	2: (* === Check loop *)
		IF NOT (MB_Lock OR MB_Start) THEN
			WHILE VarCnt<=(VARS_Max-1) AND VarSta=2 DO
				(* Check only active vars *)
				IF VARS[VarCnt].Variable<>0 THEN			(* "Variable" is a pointer to word, so if 0 no address *)
					(* Check var auto-refresh on timer checks *)
					IF VARS[VarCnt].Refresh_Time>0 AND VARS[VarCnt].Refresh_Cnt=0 THEN
						VARS[VarCnt].Refresh_Cnt:=VARS[VarCnt].Refresh_Time;
						VarSta:=3;
					END_IF
					(* Check refresh for change or request *)
					CASE VARS[VarCnt].FunCode OF
						5,6,15,16: (* Write functions *)
							IF VARS[VarCnt].Variable_Size=1 THEN
								IF VARS[VarCnt].Variable^<>VARS[VarCnt].Variable_Mirror THEN
									VARS[VarCnt].Variable_Mirror:=VARS[VarCnt].Variable^;
									VarSta:=3;
								END_IF
							ELSE
								IF VARS[VarCnt].Variable_Mirror<>0 THEN
									VARS[VarCnt].Variable_Mirror:=0;
									VarSta:=3;
								END_IF
							END_IF
						1,2,3,4: (* Read functions *)
							IF VARS[VarCnt].Variable_Mirror<>0 THEN
								VARS[VarCnt].Variable_Mirror:=0;
								VarSta:=3;
							END_IF
					END_CASE
				END_IF
				(* Process query *)
				IF VarSta=3 THEN
					MB_Lock:=TRUE;
					MB_Query.SlaveAddress:=VARS[VarCnt].SlaveAddress;
					MB_Query.FunctionCode:=VARS[VarCnt].FunCode;
					CASE VARS[VarCnt].FunCode OF
						16#5,16#6,16#F,16#10:
							MB_Query.Read_Quantity:=0;
							MB_Query.Read_StartAddress:=0;
							MB_Query.Write_StartAddress:=VARS[VarCnt].FunAddress;
							MB_Query.Write_Quantity:=VARS[VarCnt].Variable_Size;
							IF VARS[VarCnt].Variable_Size=200 THEN
								COPY_32SWAP16(VARS[VarCnt].Variable, ADR(MB_Query.Write_Data[0]));
							ELSIF VARS[VarCnt].Variable_Size>1 THEN
								MEMCPY(VARS[VarCnt].Variable, ADR(MB_Query.Write_Data[0]), 2*VARS[VarCnt].Variable_Size);
							ELSE
								MB_Query.Write_Data[0]:=VARS[VarCnt].Variable^;
							END_IF
						16#1,16#2,16#3,16#4:
							MB_Query.Read_StartAddress:=VARS[VarCnt].FunAddress;
							IF VARS[VarCnt].Variable_Size=200 THEN MB_Query.Read_Quantity:=2; ELSE		(* 200 -->> DWORD 32bits *)
							  MB_Query.Read_Quantity:=VARS[VarCnt].Variable_Size;
							END_IF
							MB_Query.Write_StartAddress:=0;
							MB_Query.Write_Quantity:=0;
					END_CASE
					VarRetry:=0;
					MB_Start:=TRUE;
				ELSE
					VarCnt:=VarCnt+1;
				END_IF
			END_WHILE
			(* Check loop completed -> no actions *)
			IF VarSta=2 THEN VarSta:=1; END_IF
		END_IF

	3: (* === Wait & process MB response *)
		IF NOT MB_Start THEN
			IF MB_MASTER.MB_Error=0 THEN
				CASE VARS[VarCnt].FunCode OF
					1,2,3,4:
						IF VARS[VarCnt].Variable_Size=200 THEN
							COPY_32SWAP16(ADR(MB_Resp.Data), VARS[VarCnt].Variable);
						ELSIF VARS[VarCnt].Variable_Size>1 THEN
							MEMCPY(ADR(MB_Resp.Data), VARS[VarCnt].Variable, 2*VARS[VarCnt].Variable_Size);
						ELSE
							VARS[VarCnt].Variable^:=MB_Resp.Data[0];
						END_IF
				END_CASE
				MB_Lock:=FALSE;
				(* Signal error recovery *)
				IF VARS_Alarm=TRUE AND VarCnt=VarAlarm THEN
					LogEv(EL_Wrn,EO_MODBUS,ID,5,'');
					VARS_Alarm:=FALSE;
				END_IF
				(* Next var *)
				VarCnt:=VarCnt+1;
				VarSta:=2;
			ELSE
				IF VarRetry<3 THEN
					VarRetry:=VarRetry+1;
					MB_Start:=TRUE;
				ELSE
					MB_Lock:=FALSE;
					(* Signal error *)
					IF VARS_Alarm=FALSE THEN
						LogEv(EL_Wrn,EO_MODBUS,ID,3,INT_TO_STRING(MB_MASTER.MB_Error));
						VARS_Alarm:=TRUE;
						VarAlarm:=VarCnt-1;
					END_IF
					(* Next var *)
					VarCnt:=VarCnt+1;
					VarSta:=2;
				END_IF
			END_IF
		END_IF

ELSE
	VarSta:=0;
END_CASE
END_ACTION

(* POU Plant_Objects/obj_HVAC_LENNOX_FGK190H2M_new, ST *)
FUNCTION_BLOCK obj_HVAC_LENNOX_FGK190H2M_new
VAR CONSTANT
	Default_SetPointCold	: WORD 	:= 220;
	Default_SetPointHeat	: WORD 	:= 190;
	Default_SetBmsTenv		: INT 	:= -999;
	Default_SetBmsRHenv		: WORD	:= 0;
	Default_SetBmsText		: INT	:= -999;
	Default_SetBmsRHext		: WORD	:= 0;
	Default_MinThrECO		: WORD 	:= 1000;
	Default_MaxThrECO		: WORD 	:= 1500;
END_VAR
VAR_INPUT
	(* Settings *)
	ID						: BYTE;
	ADDRESS					: BYTE:=31;

	(* Controls *)
	Refresh_Period			: TIME:=t#3m;
	Refresh_Auto			: BOOL:=TRUE; (* Enable automatic refresh *)
	Refresh_Now				: BOOL; 	  (* Force an immediate refresh *)

	(* HVAC inputs	*)
	SetPointColdDay			: WORD;	(* Refresh set point	*)
	SetPointHeatDay			: WORD;	(* Heat set point		*)

	SetBmsTenv				: INT	:= Default_SetBmsTenv;	(* Environment temperature set point	*)
	SetBmsRHenv				: WORD	:= Default_SetBmsRHenv;	(* Environment humidity set point	*)
	SetBmsText				: INT	:= Default_SetBmsText;	(* External temperature set point 	*)
	SetBmsRHext				: WORD	:= Default_SetBmsRHext;	(* External humidity set point 	*)

	OnOff					: BOOL;

	MinThrECO				: WORD;
	MaxThrECO				: WORD;

END_VAR
VAR_IN_OUT
	MODBUS			: obj_MODBUS;
END_VAR
VAR_OUTPUT
	(* Sono read-only tetto il mondo *)
	Data			: typ_MODBUS_HVAC_LENNOX_FGK190H2M_new;
	tmpData			: typ_MODBUS_HVAC_LENNOX_FGK190H2M_new;

	(* Status *)
	Status_Log		: BYTE;
	Status_Vis 		: DWORD;

END_VAR
VAR

	dly 		: TON := (PT:=t#5s);
	sta			: BYTE; 	(* Status *)
	retry		: BYTE;
	fModbusAlr	: BOOL;

	ModbusAlr	:	FLT_EVENT;
	Alr1		:	FLT_EVENT;
	Alr2		:	FLT_EVENT;
	Alr3		:	FLT_EVENT;
	Alr4		:	FLT_EVENT;
	Alr5		:	FLT_EVENT;
	Alr6		:	FLT_EVENT;
	Alr7		:	FLT_EVENT;

	OldAlarm1	:	WORD;
	OldAlarm2	:	WORD;
	OldAlarm3	:	WORD;
	OldAlarm4	:	WORD;
	OldAlarm5	:	WORD;
	OldAlarm6	:	WORD;
	OldAlarm7	:	WORD;

	ChangedBits	:	WORD;
	AlarmCtr	:	BYTE;

	s1			:	STRING;
END_VAR
(* Verify inputs are in the right range	*)
CheckInputs();

(* Call ModBus state machine	*)
Stm();

(* Check if an alarm occurs	*)
CheckAlarm();

IF AlarmCtr>0 THEN
	Status_Log 	:= 2;
	Status_Vis	:= COLOR_RED;
ELSE
	Status_Log	:= 0;
	Status_Vis	:= COLOR_GREEN;
END_IF
END_FUNCTION_BLOCK
ACTION AddLogData:
Logger.s1:=INSERT('&HVAC=',BYTE_TO_STRING(ID),4);
IF ID<10 THEN Logger.s1:=INSERT(Logger.s1,'0',4); END_IF

Logger.s1:=CONCAT(Logger.s1,INT_TO_STRING(Data.Tsend));					Logger.s1:=CONCAT(Logger.s1,';');
Logger.s1:=CONCAT(Logger.s1,INT_TO_STRING(Data.Treturn));				Logger.s1:=CONCAT(Logger.s1,';');
Logger.s1:=CONCAT(Logger.s1,WORD_TO_STRING(Data.AirDiffPressure));		Logger.s1:=CONCAT(Logger.s1,';');
Logger.s1:=CONCAT(Logger.s1,WORD_TO_STRING(Data.AirValve));				Logger.s1:=CONCAT(Logger.s1,';');
Logger.s1:=CONCAT(Logger.s1,WORD_TO_STRING(Data.AirGas));				Logger.s1:=CONCAT(Logger.s1,';');
Logger.s1:=CONCAT(Logger.s1,WORD_TO_STRING(Data.Triac));				Logger.s1:=CONCAT(Logger.s1,';');
Logger.s1:=CONCAT(Logger.s1,WORD_TO_STRING(Data.HWB));					Logger.s1:=CONCAT(Logger.s1,';');
Logger.s1:=CONCAT(Logger.s1,WORD_TO_STRING(Data.Humidifier));			Logger.s1:=CONCAT(Logger.s1,';');

(* Create boolean representation of status flag and convert it in string *)
(*s1:=BOOL_TO_STRING(Data.StatusFlag.0);
s1:=CONCAT(s1,BOOL_TO_STRING(Data.StatusFlag.1));
s1:=CONCAT(s1,BOOL_TO_STRING(Data.StatusFlag.2));
s1:=CONCAT(s1,BOOL_TO_STRING(Data.StatusFlag.3));
s1:=CONCAT(s1,BOOL_TO_STRING(Data.StatusFlag.4));
s1:=CONCAT(s1,BOOL_TO_STRING(Data.StatusFlag.5));
s1:=CONCAT(s1,BOOL_TO_STRING(Data.StatusFlag.6));
s1:=CONCAT(s1,BOOL_TO_STRING(Data.StatusFlag.7));
s1:=CONCAT(s1,BOOL_TO_STRING(Data.StatusFlag.8));
s1:=CONCAT(s1,BOOL_TO_STRING(Data.StatusFlag.9));
s1:=CONCAT(s1,BOOL_TO_STRING(Data.StatusFlag.10));
s1:=CONCAT(s1,BOOL_TO_STRING(Data.StatusFlag.11));
s1:=CONCAT(s1,BOOL_TO_STRING(Data.StatusFlag.12));
s1:=CONCAT(s1,BOOL_TO_STRING(Data.StatusFlag.13));*)
s1:=BOOL_TO_STRING(Data.StatusFlag.13);
s1:=CONCAT(s1,BOOL_TO_STRING(Data.StatusFlag.12));
s1:=CONCAT(s1,BOOL_TO_STRING(Data.StatusFlag.11));
s1:=CONCAT(s1,BOOL_TO_STRING(Data.StatusFlag.10));
s1:=CONCAT(s1,BOOL_TO_STRING(Data.StatusFlag.9));
s1:=CONCAT(s1,BOOL_TO_STRING(Data.StatusFlag.8));
s1:=CONCAT(s1,BOOL_TO_STRING(Data.StatusFlag.7));
s1:=CONCAT(s1,BOOL_TO_STRING(Data.StatusFlag.6));
s1:=CONCAT(s1,BOOL_TO_STRING(Data.StatusFlag.5));
s1:=CONCAT(s1,BOOL_TO_STRING(Data.StatusFlag.4));
s1:=CONCAT(s1,BOOL_TO_STRING(Data.StatusFlag.3));
s1:=CONCAT(s1,BOOL_TO_STRING(Data.StatusFlag.2));
s1:=CONCAT(s1,BOOL_TO_STRING(Data.StatusFlag.1));
s1:=CONCAT(s1,BOOL_TO_STRING(Data.StatusFlag.0));

Logger.s1:=CONCAT(Logger.s1,s1);										Logger.s1:=CONCAT(Logger.s1,';');

(* Add operation times *)
Logger.s1:=CONCAT(Logger.s1,DWORD_TO_STRING(Data.HourVent));			Logger.s1:=CONCAT(Logger.s1,';');
Logger.s1:=CONCAT(Logger.s1,DWORD_TO_STRING(Data.HourCir1Comp1));		Logger.s1:=CONCAT(Logger.s1,';');
Logger.s1:=CONCAT(Logger.s1,DWORD_TO_STRING(Data.HourCir1Comp2));		Logger.s1:=CONCAT(Logger.s1,';');
Logger.s1:=CONCAT(Logger.s1,DWORD_TO_STRING(Data.HourCir2Comp1));		Logger.s1:=CONCAT(Logger.s1,';');
Logger.s1:=CONCAT(Logger.s1,DWORD_TO_STRING(Data.HourCir2Comp2));		Logger.s1:=CONCAT(Logger.s1,';');

Logger.s1:=CONCAT(Logger.s1,BYTE_TO_STRING(Status_Log));
ADDSTRING(ADR(Logger.TData), ADR(Logger.s1), Logger.TLen);
END_ACTION
ACTION CheckAlarm:
(* Modbus alarm *)
ModbusAlr(IN:=fModbusAlr);

IF ModbusAlr.EVH THEN
	LogEv(EL_Wrn,EO_HVAC,ID,2,SEL(ModBus.MB_MASTER.MB_Error<>0,'0','1'));
	Status_Log := 1;
END_IF

IF ModbusAlr.EVL THEN Status_Log := 0; END_IF	(* If there is an alarm, "Status_Log" wil be overwritten and becomes 2 *)


(***	ALARM 1		***)
(* Verify if at least one bit has changed in register "Alarm 1"	*)
Alr1(IN:=(Data.Alarm1 <> OldAlarm1));

IF Alr1.EVH THEN
	(* Consider just bit(s) that has changed its value (indicated by a logical 1 in "ChangedBits")	*)
	ChangedBits:= Data.Alarm1 XOR OldAlarm1;

	IF ChangedBits.0 THEN
		IF Data.Alarm1.0 THEN LogEv(EL_Alarm,EO_HVAC,ID,3,'70');	AlarmCtr := AlarmCtr + 1;
		ELSE LogEv(EL_Log,EO_HVAC,ID,4,'70'); 						AlarmCtr := AlarmCtr - 1;	END_IF
	END_IF

	IF ChangedBits.1 THEN
		IF Data.Alarm1.1 THEN LogEv(EL_Alarm,EO_HVAC,ID,3,'71');	AlarmCtr := AlarmCtr + 1;
		ELSE LogEv(EL_Log,EO_HVAC,ID,4,'71'); 						AlarmCtr := AlarmCtr - 1;	END_IF
	END_IF

	IF ChangedBits.2 THEN
		IF Data.Alarm1.2 THEN LogEv(EL_Alarm,EO_HVAC,ID,3,'72');	AlarmCtr := AlarmCtr + 1;
		ELSE LogEv(EL_Log,EO_HVAC,ID,4,'72'); 						AlarmCtr := AlarmCtr - 1;	END_IF
	END_IF

	IF ChangedBits.3 THEN
		IF Data.Alarm1.3 THEN LogEv(EL_Alarm,EO_HVAC,ID,3,'9');		AlarmCtr := AlarmCtr + 1;
		ELSE LogEv(EL_Log,EO_HVAC,ID,4,'9'); 						AlarmCtr := AlarmCtr - 1;	END_IF
	END_IF

	IF ChangedBits.4 THEN
		IF Data.Alarm1.4 THEN LogEv(EL_Alarm,EO_HVAC,ID,3,'81');	AlarmCtr := AlarmCtr + 1;
		ELSE LogEv(EL_Log,EO_HVAC,ID,4,'81'); 						AlarmCtr := AlarmCtr - 1;	END_IF
	END_IF

	IF ChangedBits.5 THEN
		IF Data.Alarm1.5 THEN LogEv(EL_Alarm,EO_HVAC,ID,3,'82');	AlarmCtr := AlarmCtr + 1;
		ELSE LogEv(EL_Log,EO_HVAC,ID,4,'82'); 						AlarmCtr := AlarmCtr - 1;	END_IF
	END_IF

	IF ChangedBits.6 THEN
		IF Data.Alarm1.6 THEN LogEv(EL_Alarm,EO_HVAC,ID,3,'83');	AlarmCtr := AlarmCtr + 1;
		ELSE LogEv(EL_Log,EO_HVAC,ID,4,'83'); 						AlarmCtr := AlarmCtr - 1;	END_IF
	END_IF

	IF ChangedBits.7 THEN
		IF Data.Alarm1.7 THEN LogEv(EL_Alarm,EO_HVAC,ID,3,'85');	AlarmCtr := AlarmCtr + 1;
		ELSE LogEv(EL_Log,EO_HVAC,ID,4,'85'); 						AlarmCtr := AlarmCtr - 1;	END_IF
	END_IF

	IF ChangedBits.8 THEN
		IF Data.Alarm1.8 THEN LogEv(EL_Alarm,EO_HVAC,ID,3,'88');	AlarmCtr := AlarmCtr + 1;
		ELSE LogEv(EL_Log,EO_HVAC,ID,4,'88'); 						AlarmCtr := AlarmCtr - 1;	END_IF
	END_IF

	IF ChangedBits.9 THEN
		IF Data.Alarm1.9 THEN LogEv(EL_Alarm,EO_HVAC,ID,3,'22');	AlarmCtr := AlarmCtr + 1;
		ELSE LogEv(EL_Log,EO_HVAC,ID,4,'22'); 						AlarmCtr := AlarmCtr - 1;	END_IF
	END_IF

	IF ChangedBits.10 THEN
		IF Data.Alarm1.10 THEN LogEv(EL_Alarm,EO_HVAC,ID,3,'80');	AlarmCtr := AlarmCtr + 1;
		ELSE LogEv(EL_Log,EO_HVAC,ID,4,'80'); 						AlarmCtr := AlarmCtr - 1;	END_IF
	END_IF

	IF ChangedBits.11 THEN
		IF Data.Alarm1.11 THEN LogEv(EL_Alarm,EO_HVAC,ID,3,'73');	AlarmCtr := AlarmCtr + 1;
		ELSE LogEv(EL_Log,EO_HVAC,ID,4,'73');	 					AlarmCtr := AlarmCtr - 1;	END_IF
	END_IF

	IF ChangedBits.12 THEN
		IF Data.Alarm1.12 THEN LogEv(EL_Alarm,EO_HVAC,ID,3,'1');	AlarmCtr := AlarmCtr + 1;
		ELSE LogEv(EL_Log,EO_HVAC,ID,4,'1'); 						AlarmCtr := AlarmCtr - 1;	END_IF
	END_IF

	IF ChangedBits.13 THEN
		IF Data.Alarm1.13 THEN LogEv(EL_Alarm,EO_HVAC,ID,3,'91');	AlarmCtr := AlarmCtr + 1;
		ELSE LogEv(EL_Log,EO_HVAC,ID,4,'91'); 						AlarmCtr := AlarmCtr - 1;	END_IF
	END_IF

	IF ChangedBits.14 THEN
		IF Data.Alarm1.14 THEN LogEv(EL_Alarm,EO_HVAC,ID,3,'92');	AlarmCtr := AlarmCtr + 1;
		ELSE LogEv(EL_Log,EO_HVAC,ID,4,'92'); 						AlarmCtr := AlarmCtr - 1;	END_IF
	END_IF

	IF ChangedBits.15 THEN
		IF Data.Alarm1.15 THEN LogEv(EL_Alarm,EO_HVAC,ID,3,'99');	AlarmCtr := AlarmCtr + 1;
		ELSE LogEv(EL_Log,EO_HVAC,ID,4,'99'); 						AlarmCtr := AlarmCtr - 1;	END_IF
	END_IF

END_IF


(***	ALARM 2		***)
Alr2(IN:=(Data.Alarm2 <> OldAlarm2));

IF Alr2.EVH THEN

	ChangedBits:= Data.Alarm2 XOR OldAlarm2;

	IF ChangedBits.0 THEN
		IF Data.Alarm2.0 THEN LogEv(EL_Alarm,EO_HVAC,ID,3,'74');	AlarmCtr := AlarmCtr + 1;
		ELSE LogEv(EL_Log,EO_HVAC,ID,4,'74'); 						AlarmCtr := AlarmCtr - 1;	END_IF
	END_IF

	IF ChangedBits.1 THEN
		IF Data.Alarm2.1 THEN LogEv(EL_Alarm,EO_HVAC,ID,3,'93');	AlarmCtr := AlarmCtr + 1;
		ELSE LogEv(EL_Log,EO_HVAC,ID,4,'93'); 						AlarmCtr := AlarmCtr - 1;	END_IF
	END_IF

	IF ChangedBits.2 THEN
		IF Data.Alarm2.2 THEN LogEv(EL_Alarm,EO_HVAC,ID,3,'94');	AlarmCtr := AlarmCtr + 1;
		ELSE LogEv(EL_Log,EO_HVAC,ID,4,'94'); 						AlarmCtr := AlarmCtr - 1;	END_IF
	END_IF

	(* No bit3 for this register	*)

	IF ChangedBits.4 THEN
		IF Data.Alarm2.4 THEN LogEv(EL_Alarm,EO_HVAC,ID,3,'59');	AlarmCtr := AlarmCtr + 1;
		ELSE LogEv(EL_Log,EO_HVAC,ID,4,'59'); 						AlarmCtr := AlarmCtr - 1;	END_IF
	END_IF

	IF ChangedBits.5 THEN
		IF Data.Alarm2.5 THEN LogEv(EL_Alarm,EO_HVAC,ID,3,'56');	AlarmCtr := AlarmCtr + 1;
		ELSE LogEv(EL_Log,EO_HVAC,ID,4,'56'); 						AlarmCtr := AlarmCtr - 1;	END_IF
	END_IF

	IF ChangedBits.6 THEN
		IF Data.Alarm2.6 THEN LogEv(EL_Alarm,EO_HVAC,ID,3,'51');	AlarmCtr := AlarmCtr + 1;
		ELSE LogEv(EL_Log,EO_HVAC,ID,4,'51'); 						AlarmCtr := AlarmCtr - 1;	END_IF
	END_IF

	IF ChangedBits.7 THEN
		IF Data.Alarm2.7 THEN LogEv(EL_Alarm,EO_HVAC,ID,3,'52');	AlarmCtr := AlarmCtr + 1;
		ELSE LogEv(EL_Log,EO_HVAC,ID,4,'52'); 						AlarmCtr := AlarmCtr - 1;	END_IF
	END_IF

	(* No bit8 for this register	*)

	IF ChangedBits.9 THEN
		IF Data.Alarm2.9 THEN LogEv(EL_Alarm,EO_HVAC,ID,3,'13');	AlarmCtr := AlarmCtr + 1;
		ELSE LogEv(EL_Log,EO_HVAC,ID,4,'13'); 						AlarmCtr := AlarmCtr - 1;	END_IF
	END_IF

	IF ChangedBits.10 THEN
		IF Data.Alarm2.10 THEN LogEv(EL_Alarm,EO_HVAC,ID,3,'41');	AlarmCtr := AlarmCtr + 1;
		ELSE LogEv(EL_Log,EO_HVAC,ID,4,'41'); 						AlarmCtr := AlarmCtr - 1;	END_IF
	END_IF

	IF ChangedBits.11 THEN
		IF Data.Alarm2.11 THEN LogEv(EL_Alarm,EO_HVAC,ID,3,'11');	AlarmCtr := AlarmCtr + 1;
		ELSE LogEv(EL_Log,EO_HVAC,ID,4,'11'); 						AlarmCtr := AlarmCtr - 1;	END_IF
	END_IF

	IF ChangedBits.12 THEN
		IF Data.Alarm2.12 THEN LogEv(EL_Alarm,EO_HVAC,ID,3,'12');	AlarmCtr := AlarmCtr + 1;
		ELSE LogEv(EL_Log,EO_HVAC,ID,4,'12'); 						AlarmCtr := AlarmCtr - 1;	END_IF
	END_IF

	IF ChangedBits.13 THEN
		IF Data.Alarm2.13 THEN LogEv(EL_Alarm,EO_HVAC,ID,3,'14');	AlarmCtr := AlarmCtr + 1;
		ELSE LogEv(EL_Log,EO_HVAC,ID,4,'14'); 						AlarmCtr := AlarmCtr - 1;	END_IF
	END_IF

	IF ChangedBits.14 THEN
		IF Data.Alarm2.14 THEN LogEv(EL_Alarm,EO_HVAC,ID,3,'15');	AlarmCtr := AlarmCtr + 1;
		ELSE LogEv(EL_Log,EO_HVAC,ID,4,'15'); 						AlarmCtr := AlarmCtr - 1;	END_IF
	END_IF

	IF ChangedBits.15 THEN
		IF Data.Alarm2.15 THEN LogEv(EL_Alarm,EO_HVAC,ID,3,'16');	AlarmCtr := AlarmCtr + 1;
		ELSE LogEv(EL_Log,EO_HVAC,ID,4,'16'); 						AlarmCtr := AlarmCtr - 1;	END_IF
	END_IF

END_IF


(***	ALARM 3		***)
Alr3(IN:=(Data.Alarm3 <> OldAlarm3));

IF Alr3.EVH THEN

	ChangedBits:= Data.Alarm3 XOR OldAlarm3;

	IF ChangedBits.0 THEN
		IF Data.Alarm3.0 THEN LogEv(EL_Alarm,EO_HVAC,ID,3,'141');	AlarmCtr := AlarmCtr + 1;
		ELSE LogEv(EL_Log,EO_HVAC,ID,4,'141'); 						AlarmCtr := AlarmCtr - 1;	END_IF
	END_IF

	IF ChangedBits.1 THEN
		IF Data.Alarm3.1 THEN LogEv(EL_Alarm,EO_HVAC,ID,3,'142');	AlarmCtr := AlarmCtr + 1;
		ELSE LogEv(EL_Log,EO_HVAC,ID,4,'142'); 						AlarmCtr := AlarmCtr - 1;	END_IF
	END_IF

	IF ChangedBits.2 THEN
		IF Data.Alarm3.2 THEN LogEv(EL_Alarm,EO_HVAC,ID,3,'143');	AlarmCtr := AlarmCtr + 1;
		ELSE LogEv(EL_Log,EO_HVAC,ID,4,'143'); 						AlarmCtr := AlarmCtr - 1;	END_IF
	END_IF

	IF ChangedBits.3 THEN
		IF Data.Alarm3.3 THEN LogEv(EL_Alarm,EO_HVAC,ID,3,'144');	AlarmCtr := AlarmCtr + 1;
		ELSE LogEv(EL_Log,EO_HVAC,ID,4,'144'); 						AlarmCtr := AlarmCtr - 1;	END_IF
	END_IF

	IF ChangedBits.4 THEN
		IF Data.Alarm3.4 THEN LogEv(EL_Alarm,EO_HVAC,ID,3,'114');	AlarmCtr := AlarmCtr + 1;
		ELSE LogEv(EL_Log,EO_HVAC,ID,4,'114'); 						AlarmCtr := AlarmCtr - 1;	END_IF
	END_IF

	IF ChangedBits.5 THEN
		IF Data.Alarm3.5 THEN LogEv(EL_Alarm,EO_HVAC,ID,3,'115');	AlarmCtr := AlarmCtr + 1;
		ELSE LogEv(EL_Log,EO_HVAC,ID,4,'115'); 						AlarmCtr := AlarmCtr - 1;	END_IF
	END_IF

	IF ChangedBits.6 THEN
		IF Data.Alarm3.6 THEN LogEv(EL_Alarm,EO_HVAC,ID,3,'116');	AlarmCtr := AlarmCtr + 1;
		ELSE LogEv(EL_Log,EO_HVAC,ID,4,'116'); 						AlarmCtr := AlarmCtr - 1;	END_IF
	END_IF

	IF ChangedBits.7 THEN
		IF Data.Alarm3.7 THEN LogEv(EL_Alarm,EO_HVAC,ID,3,'117');	AlarmCtr := AlarmCtr + 1;
		ELSE LogEv(EL_Log,EO_HVAC,ID,4,'117'); 						AlarmCtr := AlarmCtr - 1;	END_IF
	END_IF

	IF ChangedBits.8 THEN
		IF Data.Alarm3.8 THEN LogEv(EL_Alarm,EO_HVAC,ID,3,'118');	AlarmCtr := AlarmCtr + 1;
		ELSE LogEv(EL_Log,EO_HVAC,ID,4,'118'); 						AlarmCtr := AlarmCtr - 1;	END_IF
	END_IF

	IF ChangedBits.9 THEN
		IF Data.Alarm3.9 THEN LogEv(EL_Alarm,EO_HVAC,ID,3,'132');	AlarmCtr := AlarmCtr + 1;
		ELSE LogEv(EL_Log,EO_HVAC,ID,4,'132'); 						AlarmCtr := AlarmCtr - 1;	END_IF
	END_IF

	IF ChangedBits.10 THEN
		IF Data.Alarm3.10 THEN LogEv(EL_Alarm,EO_HVAC,ID,3,'75');	AlarmCtr := AlarmCtr + 1;
		ELSE LogEv(EL_Log,EO_HVAC,ID,4,'75'); 						AlarmCtr := AlarmCtr - 1;	END_IF
	END_IF

	IF ChangedBits.11 THEN
		IF Data.Alarm3.11 THEN LogEv(EL_Alarm,EO_HVAC,ID,3,'102');	AlarmCtr := AlarmCtr + 1;
		ELSE LogEv(EL_Log,EO_HVAC,ID,4,'102'); 						AlarmCtr := AlarmCtr - 1;	END_IF
	END_IF

	IF ChangedBits.12 THEN
		IF Data.Alarm3.12 THEN LogEv(EL_Alarm,EO_HVAC,ID,3,'103');	AlarmCtr := AlarmCtr + 1;
		ELSE LogEv(EL_Log,EO_HVAC,ID,4,'103'); 						AlarmCtr := AlarmCtr - 1;	END_IF
	END_IF

	IF ChangedBits.13 THEN
		IF Data.Alarm3.13 THEN LogEv(EL_Alarm,EO_HVAC,ID,3,'86');	AlarmCtr := AlarmCtr + 1;
		ELSE LogEv(EL_Log,EO_HVAC,ID,4,'86'); 						AlarmCtr := AlarmCtr - 1;	END_IF
	END_IF

	IF ChangedBits.14 THEN
		IF Data.Alarm3.14 THEN LogEv(EL_Alarm,EO_HVAC,ID,3,'87');	AlarmCtr := AlarmCtr + 1;
		ELSE LogEv(EL_Log,EO_HVAC,ID,4,'87'); 						AlarmCtr := AlarmCtr - 1;	END_IF
	END_IF

	IF ChangedBits.15 THEN
		IF Data.Alarm3.15 THEN LogEv(EL_Alarm,EO_HVAC,ID,3,'101');	AlarmCtr := AlarmCtr + 1;
		ELSE LogEv(EL_Log,EO_HVAC,ID,4,'101'); 						AlarmCtr := AlarmCtr - 1;	END_IF
	END_IF

END_IF


(***	ALARM 4		***)
Alr4(IN:=(Data.Alarm4 <> OldAlarm4));

IF Alr4.EVH THEN

	ChangedBits:= Data.Alarm4 XOR OldAlarm4;

	IF ChangedBits.0 THEN
		IF Data.Alarm4.0 THEN LogEv(EL_Alarm,EO_HVAC,ID,3,'241');	AlarmCtr := AlarmCtr + 1;
		ELSE LogEv(EL_Log,EO_HVAC,ID,4,'241'); 						AlarmCtr := AlarmCtr - 1;	END_IF
	END_IF

	IF ChangedBits.1 THEN
		IF Data.Alarm4.1 THEN LogEv(EL_Alarm,EO_HVAC,ID,3,'242');	AlarmCtr := AlarmCtr + 1;
		ELSE LogEv(EL_Log,EO_HVAC,ID,4,'242'); 						AlarmCtr := AlarmCtr - 1;	END_IF
	END_IF

	IF ChangedBits.2 THEN
		IF Data.Alarm4.2 THEN LogEv(EL_Alarm,EO_HVAC,ID,3,'243');	AlarmCtr := AlarmCtr + 1;
		ELSE LogEv(EL_Log,EO_HVAC,ID,4,'243'); 						AlarmCtr := AlarmCtr - 1;	END_IF
	END_IF

	IF ChangedBits.3 THEN
		IF Data.Alarm4.3 THEN LogEv(EL_Alarm,EO_HVAC,ID,3,'244');	AlarmCtr := AlarmCtr + 1;
		ELSE LogEv(EL_Log,EO_HVAC,ID,4,'244'); 						AlarmCtr := AlarmCtr - 1;	END_IF
	END_IF

	IF ChangedBits.4 THEN
		IF Data.Alarm4.4 THEN LogEv(EL_Alarm,EO_HVAC,ID,3,'214');	AlarmCtr := AlarmCtr + 1;
		ELSE LogEv(EL_Log,EO_HVAC,ID,4,'214'); 						AlarmCtr := AlarmCtr - 1;	END_IF
	END_IF

	IF ChangedBits.5 THEN
		IF Data.Alarm4.5 THEN LogEv(EL_Alarm,EO_HVAC,ID,3,'215');	AlarmCtr := AlarmCtr + 1;
		ELSE LogEv(EL_Log,EO_HVAC,ID,4,'215'); 						AlarmCtr := AlarmCtr - 1;	END_IF
	END_IF

	IF ChangedBits.6 THEN
		IF Data.Alarm4.6 THEN LogEv(EL_Alarm,EO_HVAC,ID,3,'216');	AlarmCtr := AlarmCtr + 1;
		ELSE LogEv(EL_Log,EO_HVAC,ID,4,'216'); 						AlarmCtr := AlarmCtr - 1;	END_IF
	END_IF

	IF ChangedBits.7 THEN
		IF Data.Alarm4.7 THEN LogEv(EL_Alarm,EO_HVAC,ID,3,'217');	AlarmCtr := AlarmCtr + 1;
		ELSE LogEv(EL_Log,EO_HVAC,ID,4,'217'); 						AlarmCtr := AlarmCtr - 1;	END_IF
	END_IF

	IF ChangedBits.8 THEN
		IF Data.Alarm4.8 THEN LogEv(EL_Alarm,EO_HVAC,ID,3,'218');	AlarmCtr := AlarmCtr + 1;
		ELSE LogEv(EL_Log,EO_HVAC,ID,4,'218'); 						AlarmCtr := AlarmCtr - 1;	END_IF
	END_IF

	IF ChangedBits.9 THEN
		IF Data.Alarm4.9 THEN LogEv(EL_Alarm,EO_HVAC,ID,3,'232');	AlarmCtr := AlarmCtr + 1;
		ELSE LogEv(EL_Log,EO_HVAC,ID,4,'232'); 						AlarmCtr := AlarmCtr - 1;	END_IF
	END_IF

	IF ChangedBits.10 THEN
		IF Data.Alarm4.10 THEN LogEv(EL_Alarm,EO_HVAC,ID,3,'76');	AlarmCtr := AlarmCtr + 1;
		ELSE LogEv(EL_Log,EO_HVAC,ID,4,'76'); 						AlarmCtr := AlarmCtr - 1;	END_IF
	END_IF

	IF ChangedBits.11 THEN
		IF Data.Alarm4.11 THEN LogEv(EL_Alarm,EO_HVAC,ID,3,'202');	AlarmCtr := AlarmCtr + 1;
		ELSE LogEv(EL_Log,EO_HVAC,ID,4,'202'); 						AlarmCtr := AlarmCtr - 1;	END_IF
	END_IF

	IF ChangedBits.12 THEN
		IF Data.Alarm4.12 THEN LogEv(EL_Alarm,EO_HVAC,ID,3,'203');	AlarmCtr := AlarmCtr + 1;
		ELSE LogEv(EL_Log,EO_HVAC,ID,4,'203'); 						AlarmCtr := AlarmCtr - 1;	END_IF
	END_IF

	IF ChangedBits.13 THEN
		IF Data.Alarm4.13 THEN LogEv(EL_Alarm,EO_HVAC,ID,3,'2');	AlarmCtr := AlarmCtr + 1;
		ELSE LogEv(EL_Log,EO_HVAC,ID,4,'2'); 						AlarmCtr := AlarmCtr - 1;	END_IF
	END_IF

	IF ChangedBits.14 THEN
		IF Data.Alarm4.14 THEN LogEv(EL_Alarm,EO_HVAC,ID,3,'25');	AlarmCtr := AlarmCtr + 1;
		ELSE LogEv(EL_Log,EO_HVAC,ID,4,'25'); 						AlarmCtr := AlarmCtr - 1;	END_IF
	END_IF

	IF ChangedBits.15 THEN
		IF Data.Alarm4.15 THEN LogEv(EL_Alarm,EO_HVAC,ID,3,'26');	AlarmCtr := AlarmCtr + 1;
		ELSE LogEv(EL_Log,EO_HVAC,ID,4,'26'); 						AlarmCtr := AlarmCtr - 1;	END_IF
	END_IF

END_IF


(***	ALARM 5		***)
Alr5(IN:=(Data.Alarm5 <> OldAlarm5));

IF Alr5.EVH THEN

	ChangedBits:= Data.Alarm5 XOR OldAlarm5;

	IF ChangedBits.0 THEN
		IF Data.Alarm5.0 THEN LogEv(EL_Alarm,EO_HVAC,ID,3,'84');	AlarmCtr := AlarmCtr + 1;
		ELSE LogEv(EL_Log,EO_HVAC,ID,4,'84'); 						AlarmCtr := AlarmCtr - 1;	END_IF
	END_IF

	IF ChangedBits.1 THEN
		IF Data.Alarm5.1 THEN LogEv(EL_Alarm,EO_HVAC,ID,3,'23');	AlarmCtr := AlarmCtr + 1;
		ELSE LogEv(EL_Log,EO_HVAC,ID,4,'23'); 						AlarmCtr := AlarmCtr - 1;	END_IF
	END_IF

	IF ChangedBits.2 THEN
		IF Data.Alarm5.2 THEN LogEv(EL_Alarm,EO_HVAC,ID,3,'24');	AlarmCtr := AlarmCtr + 1;
		ELSE LogEv(EL_Log,EO_HVAC,ID,4,'24'); 						AlarmCtr := AlarmCtr - 1;	END_IF
	END_IF

	IF ChangedBits.3 THEN
		IF Data.Alarm5.3 THEN LogEv(EL_Alarm,EO_HVAC,ID,3,'32');	AlarmCtr := AlarmCtr + 1;
		ELSE LogEv(EL_Log,EO_HVAC,ID,4,'32'); 						AlarmCtr := AlarmCtr - 1;	END_IF
	END_IF

	IF ChangedBits.4 THEN
		IF Data.Alarm5.4 THEN LogEv(EL_Alarm,EO_HVAC,ID,3,'33');	AlarmCtr := AlarmCtr + 1;
		ELSE LogEv(EL_Log,EO_HVAC,ID,4,'33'); 						AlarmCtr := AlarmCtr - 1;	END_IF
	END_IF

	IF ChangedBits.5 THEN
		IF Data.Alarm5.5 THEN LogEv(EL_Alarm,EO_HVAC,ID,3,'21');	AlarmCtr := AlarmCtr + 1;
		ELSE LogEv(EL_Log,EO_HVAC,ID,4,'21'); 						AlarmCtr := AlarmCtr - 1;	END_IF
	END_IF

	IF ChangedBits.6 THEN
		IF Data.Alarm5.6 THEN LogEv(EL_Alarm,EO_HVAC,ID,3,'4');		AlarmCtr := AlarmCtr + 1;
		ELSE LogEv(EL_Log,EO_HVAC,ID,4,'4'); 						AlarmCtr := AlarmCtr - 1;	END_IF
	END_IF

	IF ChangedBits.7 THEN
		IF Data.Alarm5.7 THEN LogEv(EL_Alarm,EO_HVAC,ID,3,'5');		AlarmCtr := AlarmCtr + 1;
		ELSE LogEv(EL_Log,EO_HVAC,ID,4,'5'); 						AlarmCtr := AlarmCtr - 1;	END_IF
	END_IF

	IF ChangedBits.8 THEN
		IF Data.Alarm5.8 THEN LogEv(EL_Alarm,EO_HVAC,ID,3,'89');	AlarmCtr := AlarmCtr + 1;
		ELSE LogEv(EL_Log,EO_HVAC,ID,4,'89'); 						AlarmCtr := AlarmCtr - 1;	END_IF
	END_IF

	IF ChangedBits.9 THEN
		IF Data.Alarm5.9 THEN LogEv(EL_Alarm,EO_HVAC,ID,3,'29');	AlarmCtr := AlarmCtr + 1;
		ELSE LogEv(EL_Log,EO_HVAC,ID,4,'29'); 						AlarmCtr := AlarmCtr - 1;	END_IF
	END_IF

	IF ChangedBits.10 THEN
		IF Data.Alarm5.10 THEN LogEv(EL_Alarm,EO_HVAC,ID,3,'54');	AlarmCtr := AlarmCtr + 1;
		ELSE LogEv(EL_Log,EO_HVAC,ID,4,'54'); 						AlarmCtr := AlarmCtr - 1;	END_IF
	END_IF

	IF ChangedBits.11 THEN
		IF Data.Alarm5.11 THEN LogEv(EL_Alarm,EO_HVAC,ID,3,'31');	AlarmCtr := AlarmCtr + 1;
		ELSE LogEv(EL_Log,EO_HVAC,ID,4,'31'); 						AlarmCtr := AlarmCtr - 1;	END_IF
	END_IF

	(* No bit12 and bit13 for this register	*)

	IF ChangedBits.14 THEN
		IF Data.Alarm5.14 THEN LogEv(EL_Alarm,EO_HVAC,ID,3,'110');	AlarmCtr := AlarmCtr + 1;
		ELSE LogEv(EL_Log,EO_HVAC,ID,4,'110'); 						AlarmCtr := AlarmCtr - 1;	END_IF
	END_IF

	IF ChangedBits.15 THEN
		IF Data.Alarm5.15 THEN LogEv(EL_Alarm,EO_HVAC,ID,3,'210');	AlarmCtr := AlarmCtr + 1;
		ELSE LogEv(EL_Log,EO_HVAC,ID,4,'210'); 						AlarmCtr := AlarmCtr - 1;	END_IF
	END_IF

END_IF


(***	ALARM 6		***)
Alr6(IN:=(Data.Alarm6 <> OldAlarm6));

IF Alr6.EVH THEN

	ChangedBits:= Data.Alarm6 XOR OldAlarm6;

	IF ChangedBits.0 THEN
		IF Data.Alarm6.0 THEN LogEv(EL_Alarm,EO_HVAC,ID,3,'119');	AlarmCtr := AlarmCtr + 1;
		ELSE LogEv(EL_Log,EO_HVAC,ID,4,'119'); 						AlarmCtr := AlarmCtr - 1;	END_IF
	END_IF

	IF ChangedBits.1 THEN
		IF Data.Alarm6.1 THEN LogEv(EL_Alarm,EO_HVAC,ID,3,'129');	AlarmCtr := AlarmCtr + 1;
		ELSE LogEv(EL_Log,EO_HVAC,ID,4,'129');	 					AlarmCtr := AlarmCtr - 1;	END_IF
	END_IF

	IF ChangedBits.2 THEN
		IF Data.Alarm6.2 THEN LogEv(EL_Alarm,EO_HVAC,ID,3,'128');	AlarmCtr := AlarmCtr + 1;
		ELSE LogEv(EL_Log,EO_HVAC,ID,4,'128'); 						AlarmCtr := AlarmCtr - 1;	END_IF
	END_IF

	IF ChangedBits.3 THEN
		IF Data.Alarm6.3 THEN LogEv(EL_Alarm,EO_HVAC,ID,3,'127');	AlarmCtr := AlarmCtr + 1;
		ELSE LogEv(EL_Log,EO_HVAC,ID,4,'127'); 						AlarmCtr := AlarmCtr - 1;	END_IF
	END_IF

	IF ChangedBits.4 THEN
		IF Data.Alarm6.4 THEN LogEv(EL_Alarm,EO_HVAC,ID,3,'121');	AlarmCtr := AlarmCtr + 1;
		ELSE LogEv(EL_Log,EO_HVAC,ID,4,'121'); 						AlarmCtr := AlarmCtr - 1;	END_IF
	END_IF

	IF ChangedBits.5 THEN
		IF Data.Alarm6.5 THEN LogEv(EL_Alarm,EO_HVAC,ID,3,'122');	AlarmCtr := AlarmCtr + 1;
		ELSE LogEv(EL_Log,EO_HVAC,ID,4,'122'); 						AlarmCtr := AlarmCtr - 1;	END_IF
	END_IF

	IF ChangedBits.6 THEN
		IF Data.Alarm6.6 THEN LogEv(EL_Alarm,EO_HVAC,ID,3,'123');	AlarmCtr := AlarmCtr + 1;
		ELSE LogEv(EL_Log,EO_HVAC,ID,4,'123'); 						AlarmCtr := AlarmCtr - 1;	END_IF
	END_IF

	IF ChangedBits.7 THEN
		IF Data.Alarm6.7 THEN LogEv(EL_Alarm,EO_HVAC,ID,3,'124');	AlarmCtr := AlarmCtr + 1;
		ELSE LogEv(EL_Log,EO_HVAC,ID,4,'124'); 						AlarmCtr := AlarmCtr - 1;	END_IF
	END_IF

	IF ChangedBits.8 THEN
		IF Data.Alarm6.8 THEN LogEv(EL_Alarm,EO_HVAC,ID,3,'219');	AlarmCtr := AlarmCtr + 1;
		ELSE LogEv(EL_Log,EO_HVAC,ID,4,'219'); 						AlarmCtr := AlarmCtr - 1;	END_IF
	END_IF

	IF ChangedBits.9 THEN
		IF Data.Alarm6.9 THEN LogEv(EL_Alarm,EO_HVAC,ID,3,'229');	AlarmCtr := AlarmCtr + 1;
		ELSE LogEv(EL_Log,EO_HVAC,ID,4,'229'); 						AlarmCtr := AlarmCtr - 1;	END_IF
	END_IF

	IF ChangedBits.10 THEN
		IF Data.Alarm6.10 THEN LogEv(EL_Alarm,EO_HVAC,ID,3,'228');	AlarmCtr := AlarmCtr + 1;
		ELSE LogEv(EL_Log,EO_HVAC,ID,4,'228'); 						AlarmCtr := AlarmCtr - 1;	END_IF
	END_IF

	IF ChangedBits.11 THEN
		IF Data.Alarm6.11 THEN LogEv(EL_Alarm,EO_HVAC,ID,3,'227');	AlarmCtr := AlarmCtr + 1;
		ELSE LogEv(EL_Log,EO_HVAC,ID,4,'227'); 						AlarmCtr := AlarmCtr - 1;	END_IF
	END_IF

	IF ChangedBits.12 THEN
		IF Data.Alarm6.12 THEN LogEv(EL_Alarm,EO_HVAC,ID,3,'221');	AlarmCtr := AlarmCtr + 1;
		ELSE LogEv(EL_Log,EO_HVAC,ID,4,'221'); 						AlarmCtr := AlarmCtr - 1;	END_IF
	END_IF

	IF ChangedBits.13 THEN
		IF Data.Alarm6.13 THEN LogEv(EL_Alarm,EO_HVAC,ID,3,'222');	AlarmCtr := AlarmCtr + 1;
		ELSE LogEv(EL_Log,EO_HVAC,ID,4,'222');	 					AlarmCtr := AlarmCtr - 1;	END_IF
	END_IF

	IF ChangedBits.14 THEN
		IF Data.Alarm6.14 THEN LogEv(EL_Alarm,EO_HVAC,ID,3,'223');	AlarmCtr := AlarmCtr + 1;
		ELSE LogEv(EL_Log,EO_HVAC,ID,4,'223'); 						AlarmCtr := AlarmCtr - 1;	END_IF
	END_IF

	IF ChangedBits.15 THEN
		IF Data.Alarm6.15 THEN LogEv(EL_Alarm,EO_HVAC,ID,3,'224');	AlarmCtr := AlarmCtr + 1;
		ELSE LogEv(EL_Log,EO_HVAC,ID,4,'224'); 						AlarmCtr := AlarmCtr - 1;	END_IF
	END_IF

END_IF


(***	ALARM 7		***)
Alr7(IN:=(Data.Alarm7 <> OldAlarm7));

IF Alr7.EVH THEN

	ChangedBits:= Data.Alarm7 XOR OldAlarm7;

	IF ChangedBits.0 THEN
		IF Data.Alarm7.0 THEN LogEv(EL_Alarm,EO_HVAC,ID,3,'341');	AlarmCtr := AlarmCtr + 1;
		ELSE LogEv(EL_Log,EO_HVAC,ID,4,'341'); 						AlarmCtr := AlarmCtr - 1;	END_IF
	END_IF

	IF ChangedBits.1 THEN
		IF Data.Alarm7.1 THEN LogEv(EL_Alarm,EO_HVAC,ID,3,'342');	AlarmCtr := AlarmCtr + 1;
		ELSE LogEv(EL_Log,EO_HVAC,ID,4,'342'); 						AlarmCtr := AlarmCtr - 1;	END_IF
	END_IF

	IF ChangedBits.2 THEN
		IF Data.Alarm7.2 THEN LogEv(EL_Alarm,EO_HVAC,ID,3,'343');	AlarmCtr := AlarmCtr + 1;
		ELSE LogEv(EL_Log,EO_HVAC,ID,4,'343'); 						AlarmCtr := AlarmCtr - 1;	END_IF
	END_IF

	IF ChangedBits.3 THEN
		IF Data.Alarm7.3 THEN LogEv(EL_Alarm,EO_HVAC,ID,3,'344');	AlarmCtr := AlarmCtr + 1;
		ELSE LogEv(EL_Log,EO_HVAC,ID,4,'344'); 						AlarmCtr := AlarmCtr - 1;	END_IF
	END_IF

	IF ChangedBits.4 THEN
		IF Data.Alarm7.4 THEN LogEv(EL_Alarm,EO_HVAC,ID,3,'314');	AlarmCtr := AlarmCtr + 1;
		ELSE LogEv(EL_Log,EO_HVAC,ID,4,'314'); 						AlarmCtr := AlarmCtr - 1;	END_IF
	END_IF

	IF ChangedBits.5 THEN
		IF Data.Alarm7.5 THEN LogEv(EL_Alarm,EO_HVAC,ID,3,'315');	AlarmCtr := AlarmCtr + 1;
		ELSE LogEv(EL_Log,EO_HVAC,ID,4,'315'); 						AlarmCtr := AlarmCtr - 1;	END_IF
	END_IF

	IF ChangedBits.6 THEN
		IF Data.Alarm7.6 THEN LogEv(EL_Alarm,EO_HVAC,ID,3,'316');	AlarmCtr := AlarmCtr + 1;
		ELSE LogEv(EL_Log,EO_HVAC,ID,4,'316'); 						AlarmCtr := AlarmCtr - 1;	END_IF
	END_IF

	IF ChangedBits.7 THEN
		IF Data.Alarm7.7 THEN LogEv(EL_Alarm,EO_HVAC,ID,3,'317');	AlarmCtr := AlarmCtr + 1;
		ELSE LogEv(EL_Log,EO_HVAC,ID,4,'317'); 						AlarmCtr := AlarmCtr - 1;	END_IF
	END_IF

	IF ChangedBits.8 THEN
		IF Data.Alarm7.8 THEN LogEv(EL_Alarm,EO_HVAC,ID,3,'319');	AlarmCtr := AlarmCtr + 1;
		ELSE LogEv(EL_Log,EO_HVAC,ID,4,'319'); 						AlarmCtr := AlarmCtr - 1;	END_IF
	END_IF

	IF ChangedBits.9 THEN
		IF Data.Alarm7.9 THEN LogEv(EL_Alarm,EO_HVAC,ID,3,'329');	AlarmCtr := AlarmCtr + 1;
		ELSE LogEv(EL_Log,EO_HVAC,ID,4,'329'); 						AlarmCtr := AlarmCtr - 1;	END_IF
	END_IF

	IF ChangedBits.10 THEN
		IF Data.Alarm7.10 THEN LogEv(EL_Alarm,EO_HVAC,ID,3,'328');	AlarmCtr := AlarmCtr + 1;
		ELSE LogEv(EL_Log,EO_HVAC,ID,4,'328'); 						AlarmCtr := AlarmCtr - 1;	END_IF
	END_IF

	IF ChangedBits.11 THEN
		IF Data.Alarm7.11 THEN LogEv(EL_Alarm,EO_HVAC,ID,3,'327');	AlarmCtr := AlarmCtr + 1;
		ELSE LogEv(EL_Log,EO_HVAC,ID,4,'327'); 						AlarmCtr := AlarmCtr - 1;	END_IF
	END_IF

	IF ChangedBits.12 THEN
		IF Data.Alarm7.12 THEN LogEv(EL_Alarm,EO_HVAC,ID,3,'321');	AlarmCtr := AlarmCtr + 1;
		ELSE LogEv(EL_Log,EO_HVAC,ID,4,'321'); 						AlarmCtr := AlarmCtr - 1;	END_IF
	END_IF

	IF ChangedBits.13 THEN
		IF Data.Alarm7.13 THEN LogEv(EL_Alarm,EO_HVAC,ID,3,'322');	AlarmCtr := AlarmCtr + 1;
		ELSE LogEv(EL_Log,EO_HVAC,ID,4,'322'); 						AlarmCtr := AlarmCtr - 1;	END_IF
	END_IF

	IF ChangedBits.14 THEN
		IF Data.Alarm7.14 THEN LogEv(EL_Alarm,EO_HVAC,ID,3,'323');	AlarmCtr := AlarmCtr + 1;
		ELSE LogEv(EL_Log,EO_HVAC,ID,4,'323'); 						AlarmCtr := AlarmCtr - 1;	END_IF
	END_IF

	IF ChangedBits.15 THEN
		IF Data.Alarm7.15 THEN LogEv(EL_Alarm,EO_HVAC,ID,3,'324');	AlarmCtr := AlarmCtr + 1;
		ELSE LogEv(EL_Log,EO_HVAC,ID,4,'324'); 						AlarmCtr := AlarmCtr - 1;	END_IF
	END_IF

END_IF
END_ACTION
ACTION CheckInputs:
(* If value of variables are out of admissible range, set default value as stated in the manual	*)
IF SetPointColdDay<80 OR SetPointColdDay>350 THEN SetPointColdDay := Default_SetPointCold; END_IF
IF SetPointHeatDay<80 OR SetPointHeatDay>350 THEN SetPointHeatDay := Default_SetPointHeat; END_IF

IF SetBmsTenv<-999 OR SetBmsTenv>999 THEN SetBmsTenv := Default_SetBmsTenv; END_IF
IF SetBmsRHenv<0 OR SetBmsRHenv>1000 THEN SetBmsRHenv := Default_SetBmsRHenv; END_IF
IF SetBmsText<-999 OR SetBmsText>999 THEN SetBmsText := Default_SetBmsText; END_IF
IF SetBmsRHext<0 OR SetBmsRHext>1000 THEN SetBmsRHext := Default_SetBmsRHext; END_IF

IF MinThrECO<0 OR MinThrECO>2000 THEN MinThrECO := Default_MinThrECO; END_IF
IF MaxThrECO<0 OR MaxThrECO>2000 THEN MaxThrECO := Default_MaxThrECO; END_IF
END_ACTION
ACTION Stm:
CASE sta OF
	0: (* === Wait update signals *)
		dly(IN:=NOT (dly.Q OR Refresh_Now OR (NOT Refresh_Auto)));
		IF dly.Q OR Refresh_Now THEN
			dly.PT := Refresh_Period;
			Refresh_Now := FALSE;

			retry := 0;
			sta := 1;
		END_IF

	1: (* === Start update when MB is free *)
		IF NOT (MODBUS.MB_Lock OR MODBUS.MB_Start) THEN

			MODBUS.MB_Lock := TRUE;

			MODBUS.MB_Query.SlaveAddress		:= ADDRESS;
			MODBUS.MB_Query.FunctionCode		:= 16#03;
			MODBUS.MB_Query.Read_StartAddress	:= 36;
			MODBUS.MB_Query.Read_Quantity		:= 16;

			MODBUS.MB_Start := TRUE;
			sta := 2;
		END_IF

	2:
		IF NOT MODBUS.MB_Start THEN
			IF MODBUS.MB_MASTER.MB_Error<>MB_NO_ERROR OR MODBUS.MB_Resp.Error<>0 THEN
				sta:=100;
			ELSE

				tmpData.AlarmCode			:= MODBUS.MB_Resp.Data[0];
				tmpData.Tenv				:= WORD_TO_INT(MODBUS.MB_Resp.Data[1]);
				tmpData.Text				:= WORD_TO_INT(MODBUS.MB_Resp.Data[2]);
				tmpData.Tsend				:= WORD_TO_INT(MODBUS.MB_Resp.Data[3]);
				tmpData.Treturn				:= WORD_TO_INT(MODBUS.MB_Resp.Data[4]);
				tmpData.RH_env				:= MODBUS.MB_Resp.Data[5];
				tmpData.AH_env				:= MODBUS.MB_Resp.Data[6];
				tmpData.RH_ext				:= MODBUS.MB_Resp.Data[7];
				tmpData.AH_ext				:= MODBUS.MB_Resp.Data[8];
				tmpData.AirDiffPressure		:= MODBUS.MB_Resp.Data[9];
				tmpData.CO2_ppm				:= MODBUS.MB_Resp.Data[10];
				tmpData.AirValve			:= MODBUS.MB_Resp.Data[11];
				tmpData.AirGas				:= MODBUS.MB_Resp.Data[12];
				tmpData.Triac				:= MODBUS.MB_Resp.Data[13];
				tmpData.HWB					:= MODBUS.MB_Resp.Data[14];
				tmpData.Humidifier			:= MODBUS.MB_Resp.Data[15];

				MODBUS.MB_Query.SlaveAddress		:= ADDRESS;
				MODBUS.MB_Query.FunctionCode		:= 16#03;
				MODBUS.MB_Query.Read_StartAddress	:= 62;
				MODBUS.MB_Query.Read_Quantity		:= 10;

				MODBUS.MB_Start := TRUE;
				sta := 3;

			END_IF
		END_IF

	3:
		IF NOT MODBUS.MB_Start THEN
			IF MODBUS.MB_MASTER.MB_Error<>MB_NO_ERROR OR MODBUS.MB_Resp.Error<>0 THEN
				sta:=100;
			ELSE

				tmpData.HourVent 		:= BUILD_16TO32(ADR(MODBUS.MB_Resp.Data[0]));
				tmpData.HourCir1Comp1 	:= BUILD_16TO32(ADR(MODBUS.MB_Resp.Data[2]));
				tmpData.HourCir1Comp2 	:= BUILD_16TO32(ADR(MODBUS.MB_Resp.Data[4]));
				tmpData.HourCir2Comp1 	:= BUILD_16TO32(ADR(MODBUS.MB_Resp.Data[6]));
				tmpData.HourCir2Comp2	:= BUILD_16TO32(ADR(MODBUS.MB_Resp.Data[8]));

				MODBUS.MB_Query.SlaveAddress		:= ADDRESS;
				MODBUS.MB_Query.FunctionCode		:= 16#03;
				MODBUS.MB_Query.Read_StartAddress	:= 74;
				MODBUS.MB_Query.Read_Quantity		:= 7;

				MODBUS.MB_Start := TRUE;
				sta := 4;

			END_IF
		END_IF

	4:
		IF NOT MODBUS.MB_Start THEN
			IF MODBUS.MB_MASTER.MB_Error<>MB_NO_ERROR OR MODBUS.MB_Resp.Error<>0 THEN
				sta:=100;
			ELSE
				tmpData.Alarm1	:= MODBUS.MB_Resp.Data[0];
				tmpData.Alarm2	:= MODBUS.MB_Resp.Data[1];
				tmpData.Alarm3	:= MODBUS.MB_Resp.Data[2];
				tmpData.Alarm4	:= MODBUS.MB_Resp.Data[3];
				tmpData.Alarm5	:= MODBUS.MB_Resp.Data[4];
				tmpData.Alarm6	:= MODBUS.MB_Resp.Data[5];
				tmpData.Alarm7	:= MODBUS.MB_Resp.Data[6];

				MODBUS.MB_Query.SlaveAddress		:= ADDRESS;
				MODBUS.MB_Query.FunctionCode		:= 16#03;
				MODBUS.MB_Query.Read_StartAddress	:= 134;
				MODBUS.MB_Query.Read_Quantity		:= 16;

				MODBUS.MB_Start := TRUE;
				sta := 10;
			END_IF
		END_IF

	(* 	WRITE	*)
	10:
		IF NOT MODBUS.MB_Start THEN
			IF MODBUS.MB_MASTER.MB_Error<>MB_NO_ERROR OR MODBUS.MB_Resp.Error<>0 THEN
				sta:=100;
			ELSE
				tmpData.StatusFlag.0 := WORD_TO_BOOL(MODBUS.MB_Resp.Data[0]);
				tmpData.StatusFlag.1 := WORD_TO_BOOL(MODBUS.MB_Resp.Data[1]);
				tmpData.StatusFlag.2 := WORD_TO_BOOL(MODBUS.MB_Resp.Data[2]);
				tmpData.StatusFlag.3 := WORD_TO_BOOL(MODBUS.MB_Resp.Data[3]);
				tmpData.StatusFlag.4 := WORD_TO_BOOL(MODBUS.MB_Resp.Data[4]);
				tmpData.StatusFlag.5 := WORD_TO_BOOL(MODBUS.MB_Resp.Data[5]);
				tmpData.StatusFlag.6 := WORD_TO_BOOL(MODBUS.MB_Resp.Data[6]);
				tmpData.StatusFlag.7 := WORD_TO_BOOL(MODBUS.MB_Resp.Data[7]);
				tmpData.StatusFlag.8 := WORD_TO_BOOL(MODBUS.MB_Resp.Data[8]);
				tmpData.StatusFlag.9 := WORD_TO_BOOL(MODBUS.MB_Resp.Data[9]);
				tmpData.StatusFlag.10 := WORD_TO_BOOL(MODBUS.MB_Resp.Data[10]);
				tmpData.StatusFlag.11 := WORD_TO_BOOL(MODBUS.MB_Resp.Data[11]);
				tmpData.StatusFlag.12 := WORD_TO_BOOL(MODBUS.MB_Resp.Data[12]);
				tmpData.StatusFlag.13 := WORD_TO_BOOL(MODBUS.MB_Resp.Data[13]);

				MODBUS.MB_Query.FunctionCode 		:= 16#10;
				MODBUS.MB_Query.Write_StartAddress	:= 1;
				MODBUS.MB_Query.Write_Quantity		:= 3;
				MODBUS.MB_Query.Write_Data[0] 		:= 1000;    			(* Fixed value to refresh HVAC watchdog (the unit decreas this value
																		   by 5 every 5s. If it reaches 0, an internal error is triggered	*)
				MODBUS.MB_Query.Write_Data[1] 		:= SetPointColdDay;
				MODBUS.MB_Query.Write_Data[2] 		:= SetPointHeatDay;

				MODBUS.MB_Start := TRUE;
				sta := 11;

			END_IF
		END_IF


	11:
		IF NOT MODBUS.MB_Start THEN
			IF MODBUS.MB_MASTER.MB_Error<>MB_NO_ERROR OR MODBUS.MB_Resp.Error<>0 THEN
				sta:=100;
			ELSE

				MODBUS.MB_Query.FunctionCode 		:= 16#10;
				MODBUS.MB_Query.Write_StartAddress	:= 20;
				MODBUS.MB_Query.Write_Quantity		:= 4;
				MODBUS.MB_Query.Write_Data[0]		:= INT_TO_WORD(SetBmsTenv);
				MODBUS.MB_Query.Write_Data[1]		:= SetBmsRHenv;
				MODBUS.MB_Query.Write_Data[2]		:= INT_TO_WORD(SetBmsText);
				MODBUS.MB_Query.Write_Data[3]		:= SetBmsRHext;

				MODBUS.MB_Start := TRUE;
				sta := 12;

			END_IF
		END_IF

	12:
		IF NOT MODBUS.MB_Start THEN
			IF MODBUS.MB_MASTER.MB_Error<>MB_NO_ERROR OR MODBUS.MB_Resp.Error<>0 THEN
				sta:=100;
			ELSE

				MODBUS.MB_Query.FunctionCode		:= 16#10;
				MODBUS.MB_Query.Write_StartAddress	:= 84;
				MODBUS.MB_Query.Write_Quantity		:= 16#1;
				MODBUS.MB_Query.Write_Data[0]		:= BOOL_TO_WORD(OnOff);

				MODBUS.MB_Start := TRUE;
				sta := 13;
			END_IF
		END_IF

	13:
		IF NOT MODBUS.MB_Start THEN
			IF MODBUS.MB_MASTER.MB_Error<>MB_NO_ERROR OR MODBUS.MB_Resp.Error<>0 THEN
				sta:=100;
			ELSE

				MODBUS.MB_Query.FunctionCode		:= 16#10;
				MODBUS.MB_Query.Write_StartAddress	:= 187;
				MODBUS.MB_Query.Write_Quantity		:= 2;
				MODBUS.MB_Query.Write_Data[0]		:= MinThrECO;
				MODBUS.MB_Query.Write_Data[1]		:= MaxThrECO;

				MODBUS.MB_Start := TRUE;
				sta := 14;
			END_IF
		END_IF


	14:	IF NOT MODBUS.MB_Start THEN
			IF MODBUS.MB_MASTER.MB_Error<>MB_NO_ERROR OR MODBUS.MB_Resp.Error<>0 THEN
				sta:=100;
			ELSE
				(* Copy temporary read data *)
				MEMCPY(ADR(tmpData), ADR(Data), SIZEOF(Data));

				fModbusAlr := FALSE;
				MODBUS.MB_Lock := FALSE;
				sta := 0;
			END_IF
		END_IF


	100: (* === Check MODBUS error *)
		(* Release MODBUS *)
		MODBUS.MB_Lock := FALSE;

		(* Retries *)
		retry := retry+1;

		IF retry>3 THEN
			retry := 0;

			(* Signal event *)
			IF Status_Log<>2 THEN
				LogEv(EL_Alarm,EO_HVAC,ID,2,SEL(ModBus.MB_MASTER.MB_Error<>0,'0','1'));
			END_IF
			fModbusAlr := TRUE;
		END_IF

		sta := 0;

ELSE
	sta := 0;
END_CASE
END_ACTION

(* POU Plant_Objects/obj_LUXM, ST *)
FUNCTION_BLOCK obj_LUXM
(* === Metered ON/OFF Illumination Point ===
   Failure detection:
   Statistic data:
   
   - Come identifico l'assenza del nodo?? (Rele non funzionante/non alimentato)
   - Acquisizione carico dopo accensione?? Dati carico in NVM!
   
   v1.0[07/05/15] - Create
*)
VAR_INPUT
	(* Settings *)
	ID				: BYTE;
	(* Controls *)
	CTRL_MODE		: INT;  (* 0:MAN OFF, -1:MAN-ON,
							   -2:KEY-ON, -3:KEY-OFF, -4:DAY, -5:NIGHT,
							   N>0:Nsec-TIMER *)
	CTRL_TRIG		: BOOL; (* Trigger for timer start *)
	CTRL_KEY		: BOOL; (* External KEY control input *)
	CTRL_SENS		: BOOL; (* External dark sensor input [1:Dark] *)
	CTRL_EXTON		: BOOL; (* External forced activation *)
	(* Physical inputs *)
	REL_ST			: BOOL; (* Status feedback *)
	REL_V			: WORD; (* [E-1 V] Voltage *)
	REL_A			: WORD; (* [E-1 A] Current *)
	REL_ALM			: WORD; (* Error status [0:OK, 1:Disconnected, 2:LoadLOW, 3:LoadHIGH, 4:Overload, 5:ControlFAIL] *)
	REL_TEMP		: INT;  (* [E-1 °C] Temperature *)
	REL_TON			: DWORD;(* [sec] External working time counter *)  
	(* Persistent *)(*
	WORKINGTIME		: POINTER TO DWORD; (* [sec] Internal working time counter *)
	POWERONCYCLES	: POINTER TO DWORD; (* Internal counter of power-on cycles *)
	ENERGYCOUNTER	: POINTER TO DWORD; (* [E-1 kWh] Internal energy counter *)
	ENERGYCOUNTER_T : POINTER TO DWORD; (* Temporary energy in E-2*Wsec *)*)
END_VAR
VAR_IN_OUT
	WORKINGTIME		: DWORD; (* [sec] Internal working time counter *)
	POWERONCYCLES	: DWORD; (* Internal counter of power-on cycles *)
	ENERGYCOUNTER	: DWORD; (* [E-1 kWh] Internal energy counter *)
	ENERGYCOUNTER_T : DWORD; (* Temporary energy in E-2*Wsec *)
END_VAR
VAR_OUTPUT
	(* Physical outputs *)
	REL_EN			: BOOL;	(* Control output *)
	(* Status *)
	Status_Log		: BYTE;
	Status_Vis 		: DWORD;
END_VAR
VAR
	TickTimer		: TON := ( PT:=T#1S );
	TrigTimer		: TOF;
	sREL_EN			: FLT_EVENT;
	sREL_ALM		: WORD:=16#FFFF;
	chkREL_ST		: FLT_TIME := ( TTAP:=T#20S, INITEV:=FALSE );
END_VAR
(* Trig timer *)
TrigTimer(IN:=CTRL_TRIG);

(* Control logic *)
IF CTRL_EXTON THEN
	REL_EN:=TRUE;
ELSE
	CASE CTRL_MODE OF
		 0: REL_EN:=FALSE;
		-1: REL_EN:=TRUE;
		-2: REL_EN:=CTRL_KEY;
		-3: REL_EN:=NOT CTRL_KEY;
		-4: REL_EN:=CTRL_SENS;
		-5: REL_EN:=NOT CTRL_SENS;
	ELSE
		IF CTRL_MODE>0 THEN
			REL_EN:=TrigTimer.Q;
			TrigTimer.PT:=T#1S*CTRL_MODE;
		ELSE
			REL_EN:=FALSE;
		END_IF
	END_CASE
END_IF

(* Temporary energy counter *)
TickTimer(IN:=NOT TickTimer.Q);
IF TickTimer.Q AND REL_EN THEN
	WORKINGTIME:=WORKINGTIME+1;
	ENERGYCOUNTER_T:=ENERGYCOUNTER_T+REL_V*REL_A;
	IF ENERGYCOUNTER_T>36000000 THEN
		ENERGYCOUNTER_T:=ENERGYCOUNTER_T-36000000;
		ENERGYCOUNTER:=ENERGYCOUNTER+1;		
	END_IF
END_IF

(* Generate status events *)
sREL_EN(IN:=REL_EN);
IF sREL_EN.EVL THEN LogEv(EL_Log,EO_LUXM,ID,2,''); END_IF
IF sREL_EN.EVH THEN LogEv(EL_Log,EO_LUXM,ID,3,''); POWERONCYCLES:=POWERONCYCLES+1; END_IF

(* Check status feedback *)
chkREL_ST(IN:=(REL_ST<>REL_EN));
IF chkREL_ST.EVH THEN LogEv(EL_Alarm,EO_LUXM,ID,9,''); END_IF
IF chkREL_ST.EVL AND sREL_ALM=0 THEN LogEv(EL_Log,EO_LUXM,ID,1,''); END_IF

(* Check controller alarm *)
IF sREL_ALM<>REL_ALM THEN
	CASE REL_ALM OF
		0: IF NOT chkREL_ST.OUT THEN LogEv(EL_Log,EO_LUXM,ID,1,''); END_IF
		1: LogEv(EL_Alarm,EO_LUXM,ID,6,'');
		2: LogEv(EL_Wrn  ,EO_LUXM,ID,4,WORD_TO_STRING(REL_A));
		3: LogEv(EL_Wrn  ,EO_LUXM,ID,5,WORD_TO_STRING(REL_A));
		4: LogEv(EL_Alarm,EO_LUXM,ID,7,WORD_TO_STRING(REL_A));
		5: LogEv(EL_Alarm,EO_LUXM,ID,8,'');
	END_CASE
	sREL_ALM:=REL_ALM;
END_IF

(* Status color *)
   IF REL_ALM=1 OR REL_ALM>3 OR chkREL_ST.OUT	THEN Status_Log:=2; Status_Vis:=COLOR_RED;
ELSIF REL_ALM<>0								THEN Status_Log:=1; Status_Vis:=COLOR_YELLOW;
                  	   							ELSE Status_Log:=0; Status_Vis:=SEL(REL_EN,COLOR_GREEN_OFF,COLOR_GREEN);
END_IF
END_FUNCTION_BLOCK
ACTION AddLogData:
Logger.s1:=INSERT('&LUXM=',BYTE_TO_STRING(ID),5);
IF ID<10 THEN Logger.s1:=INSERT(Logger.s1,'0',5); END_IF

Logger.s1:=CONCAT(Logger.s1,WORD_TO_STRING(REL_V));				Logger.s1:=CONCAT(Logger.s1,';');
Logger.s1:=CONCAT(Logger.s1,WORD_TO_STRING(REL_A));				Logger.s1:=CONCAT(Logger.s1,';');
Logger.s1:=CONCAT(Logger.s1,DWORD_TO_STRING(ENERGYCOUNTER));	Logger.s1:=CONCAT(Logger.s1,';');
Logger.s1:=CONCAT(Logger.s1,DWORD_TO_STRING(WORKINGTIME));		Logger.s1:=CONCAT(Logger.s1,';');
Logger.s1:=CONCAT(Logger.s1,DWORD_TO_STRING(POWERONCYCLES));	Logger.s1:=CONCAT(Logger.s1,';');
Logger.s1:=CONCAT(Logger.s1,INT_TO_STRING(REL_TEMP));			Logger.s1:=CONCAT(Logger.s1,';');

Logger.s1:=CONCAT(Logger.s1,BYTE_TO_STRING(Status_Log));
ADDSTRING(ADR(Logger.TData), ADR(Logger.s1), Logger.TLen);
END_ACTION
ACTION StatReset:
(* Reset statistic counters *)
WORKINGTIME:=0;
POWERONCYCLES:=0;
ENERGYCOUNTER:=0;
END_ACTION

(* POU Plant_Objects/obj_LUXP, ST *)
FUNCTION_BLOCK obj_LUXP
(* === Metered ON/OFF Illumination Point ===
   Failure detection:
   Statistic data:
   
   - Come identifico l'assenza del nodo?? (Rele non funzionante/non alimentato)
   - Acquisizione carico dopo accensione?? Dati carico in NVM!
   
   v1.0[07/05/15] - Create
*)
VAR CONSTANT
	MANUAL			: BYTE := 0;
	AUTOMATIC		: BYTE := 1;
	SCHEDULED		: BYTE := 2;
END_VAR
VAR_INPUT
	(* Settings *)
	ID				: BYTE;
	(* Controls *)
	CTRL_MODE		: BYTE;  (* 0 : MANUAL, (human) user manage the lux						->	HIGHEST PRIORITY
							    1 : AUTO, external device/sensor manage the lux				->	MID PRIORITY
							    2 : SCHEDULED, scheduled profile with crono manage the lux	->	LOWEST PRIORITY
							  *)

	CTRL_KEY		: BOOL := FALSE; (* External KEY control input *)
	KEY_DEV			: BOOL := TRUE;			 (* 0: key as deviator, changes output state every time, 1: key as latch switch, 2: key as auto/manual selector *)
	CTRL_EXT_DS		: BOOL := FALSE; (* External DEVICE/SENSOR input *)
	CTRL_CRON		: BOOL := FALSE; (* External forced activation *)

	(* Conditional event *)
	CTRL_COND		: typ_Condition;
	OUT_ST_SINGLE	: BOOL;			 (* External output status signal relative to this lux available or not *)
	CTRL_MANUAL		: BOOL := FALSE;

	(* Physical inputs *)
	OUT_ST			: BOOL; (* Status feedback *)

END_VAR
VAR_IN_OUT
	WORKINGTIME		: DWORD; (* [sec] Internal working time counter *)
	POWERONCYCLES	: DWORD; (* Internal counter of power-on cycles *)
END_VAR
VAR_OUTPUT
	(* Physical outputs *)
	OUT_EN			: BOOL;	(* Control output *)
	(* Status *)
	Status_Log		: BYTE;
	Status_Vis 		: DWORD;
END_VAR
VAR
	InitOK			: BOOL;
	CTRL_MODE_Default: BYTE;
	Force			: BOOL := FALSE;		(* Force output to a value without considering its normal operation	*)

	KeyPress		: FLT_KEY 	:= (INITEV:=FALSE, TTAP:=T#5ms); (*FLT_TIME 	:= (INITEV:=FALSE, TTAP:=T#5ms);*)
	AutoEn			: FLT_TAP	:= (INITEV:=FALSE);
	sOUT_EN			: FLT_EVENT;

	TickTimer		: TON := ( PT:=T#1s );
	chkOUT_ST		: FLT_TIME := ( TTAP:=T#5s, INITEV:=FALSE );

	actualTime		: STRING;

END_VAR
IF NOT InitOK THEN
	(* First time read the CTRL_MODE setted by the programmer in the global variables definition *)
	CTRL_MODE_Default := CTRL_MODE;
	InitOK := TRUE;
END_IF

(* Check if one or more conditional events are setted for this LUX *)
Condition();

CASE CTRL_MODE OF

	MANUAL:	(* Lux switching is managed by user	*)

		KeyPress(IN:=CTRL_KEY);

		IF KEY_DEV THEN
			IF KeyPress.EVH THEN OUT_EN := NOT OUT_EN; END_IF	(* Toggle output *)
		ELSE
			IF KeyPress.EVH OR KeyPress.EVL THEN OUT_EN := CTRL_KEY; END_IF
		END_IF


	AUTOMATIC:	(* Lux managed by an external device/sensor	*)

		KeyPress(IN:=CTRL_KEY);
		(* If a change in the key state has occured, switch to manual mode	*)
		IF KEY_DEV THEN
			IF KeyPress.EVH THEN
				OUT_EN := NOT OUT_EN; 	(* Toggle output *)
				CTRL_MODE := MANUAL;
			END_IF
		ELSE
			IF KeyPress.EVH OR KeyPress.EVL THEN
				OUT_EN := CTRL_KEY;
				CTRL_MODE := MANUAL;
			END_IF
		END_IF

		IF CTRL_MODE<>MANUAL THEN
			(* If not Forced keep automatic control *)
			IF NOT Force THEN
				(* Automatic mode *)
				AutoEn(IN:=CTRL_EXT_DS);

				IF AutoEn.EVH OR AutoEn.EVL THEN OUT_EN := NOT OUT_EN; END_IF
			END_IF
		END_IF

	SCHEDULED:
		(* Check if key has changed its state	*)
		KeyPress(IN:=CTRL_KEY);

		IF KEY_DEV THEN
			IF KeyPress.EVH THEN
				OUT_EN := NOT OUT_EN; 	(* Toggle output *)
				CTRL_MODE := MANUAL;
			END_IF
		ELSE
			IF KeyPress.EVH OR KeyPress.EVL THEN
				OUT_EN := CTRL_KEY;
				CTRL_MODE := MANUAL;
			END_IF
		END_IF

		IF CTRL_MODE<>MANUAL THEN
			(* If not forced keep normal control *)
			IF NOT Force THEN
				(* Check if external control device has changed its state	*)
				AutoEn(IN:=CTRL_EXT_DS);
	
				IF AutoEn.EVH OR AutoEn.EVL THEN
					CTRL_MODE := AUTOMATIC;
					OUT_EN := NOT OUT_EN;
				ELSE
					(* Scheduled mode	*)
					OUT_EN := CTRL_CRON;
				END_IF
			END_IF
		END_IF

END_CASE

IF CTRL_MANUAL THEN OUT_EN := TRUE; END_IF

(* Temporary energy counter *)
TickTimer(IN:=NOT TickTimer.Q);
IF (TickTimer.Q AND OUT_EN) THEN WORKINGTIME:=WORKINGTIME+1; END_IF

(* Generate status events *)
sOUT_EN(IN:=OUT_EN);
IF sOUT_EN.EVL THEN LogEv(EL_Log,EO_LUXM,ID,2,''); END_IF
IF sOUT_EN.EVH THEN LogEv(EL_Log,EO_LUXM,ID,3,''); POWERONCYCLES:=POWERONCYCLES+1; END_IF

(* Check status feedback *)
IF OUT_ST_SINGLE THEN chkOUT_ST(IN:=(OUT_ST<>OUT_EN));	(* External status feedback input available *)
ELSE chkOUT_ST(IN:=OUT_ST);						(* No external status feedback *)
END_IF
IF chkOUT_ST.EVH THEN LogEv(EL_Alarm,EO_LUXM,ID,9,''); END_IF
IF chkOUT_ST.EVL THEN LogEv(EL_Log,EO_LUXM,ID,1,''); END_IF

(* Status color *)
IF chkOUT_ST.OUT	THEN Status_Log:=2; Status_Vis:=COLOR_RED;
ELSE Status_Log:=0; Status_Vis:=SEL(OUT_EN,COLOR_GREEN_OFF,COLOR_GREEN);
END_IF
END_FUNCTION_BLOCK
ACTION AddLogData:
Logger.s1:=INSERT('&LUXM=',BYTE_TO_STRING(ID),5);
IF ID<10 THEN Logger.s1:=INSERT(Logger.s1,'0',5); END_IF

Logger.s1:=CONCAT(Logger.s1,BOOL_TO_STRING(OUT_EN));			Logger.s1:=CONCAT(Logger.s1,';');
Logger.s1:=CONCAT(Logger.s1,DWORD_TO_STRING(WORKINGTIME));		Logger.s1:=CONCAT(Logger.s1,';');
Logger.s1:=CONCAT(Logger.s1,DWORD_TO_STRING(POWERONCYCLES));	Logger.s1:=CONCAT(Logger.s1,';');

Logger.s1:=CONCAT(Logger.s1,BYTE_TO_STRING(Status_Log));
ADDSTRING(ADR(Logger.TData), ADR(Logger.s1), Logger.TLen);
END_ACTION
ACTION Condition:
CASE CTRL_COND.Enable OF

	0:	(* NO CONDITION	*)
		;

	1:	(* BOOLEAN CONDITION - Trig On *)
		IF CTRL_COND.OnIN=CTRL_COND.OnValue THEN OUT_EN:=TRUE; END_IF

	2:	(* BOOLEAN CONDITION - Trig Off *)
		IF CTRL_COND.OffIN=CTRL_COND.OffValue THEN OUT_EN:=FALSE; END_IF

	3:	(* BOOLEAN CONDITION - Trig On and Off *)
		IF (OUT_EN=FALSE AND CTRL_COND.OnIN=CTRL_COND.OnValue) THEN OUT_EN:=TRUE; END_IF
		IF (OUT_EN=TRUE AND CTRL_COND.OffIN=CTRL_COND.OffValue) THEN OUT_EN:=FALSE; END_IF

	4: 	(* TIME of DAY - Trig On *)
		actualTime := MID(STR:=Sys.Time_LogString, LEN:=5, POS:=12);		(* Check if time of the day reached *)

		IF (OUT_EN=FALSE AND actualTime>=TOD_TO_STRING(CTRL_COND.OnTime)) THEN OUT_EN:=TRUE; END_IF

	5: 	(* TIME of DAY - Trig Off *)
		actualTime := MID(STR:=Sys.Time_LogString, LEN:=5, POS:=12);

		IF (OUT_EN=TRUE AND actualTime>=TOD_TO_STRING(CTRL_COND.OffTime)) THEN
			OUT_EN:= FALSE;
			Force := TRUE;
		END_IF

		IF actualTime>='08:00' THEN Force := FALSE; END_IF	(* Release force and restore normal working *)

END_CASE
END_ACTION
ACTION RestoreMode:
CTRL_MODE := CTRL_MODE_Default;
END_ACTION
ACTION StatReset:
(* Reset statistic counters *)
WORKINGTIME:=0;
POWERONCYCLES:=0;
END_ACTION

(* POU Plant_Objects/obj_MODBUS_FRER_QUBOH, ST *)
FUNCTION_BLOCK obj_MODBUS_FRER_QUBOH
(* === MODBUS ELECTRICITY CONTABILIZER ABB ===
   v1.0[20/08/15] - Versioning
*)
VAR CONSTANT
	WAIT_STATE		:	BYTE := 0;
	START_READ		:	BYTE := 1;
	READ_1			:	BYTE := 2;
	READ_2			:	BYTE := 3;
	READ_3			:	BYTE := 4;
	READ_4			:	BYTE := 5;
	READ_5			:	BYTE := 6;
	END_READ		:	BYTE := 7;

	ERROR_STATE		:	BYTE := 100;
END_VAR
VAR_INPUT
	ID				:	BYTE;
	Address			:	BYTE;

	Refresh_Period	: 	TIME:=t#3m;
	(* Controls *)
	Refresh_Auto	: 	BOOL:=TRUE; (* Enable automatic refresh *)
	Refresh_Now		:	BOOL; 	  (* Force an immediate refresh *)
END_VAR
VAR_IN_OUT
	ModBus		:	obj_MODBUS;
END_VAR
VAR_OUTPUT
	Status_Log	:	WORD;
	Status_Vis	:	DWORD;
END_VAR
VAR
	Data		:	typ_MODBUS_FRER_QUBOH;

	WH_3P		:	DWORD;		(* E-1 kWh *)
	VARH_3P		:	DWORD;		(* E-1 kVArh *)

	dly 		: 	TON := (PT:=t#5s);
	state		: 	BYTE; 	(* Status *)
	retry		: 	BYTE;
END_VAR
CASE state OF

	WAIT_STATE: (* === Wait update signals *)
		dly(IN:=NOT (dly.Q OR Refresh_Now OR (NOT Refresh_Auto)));
		IF dly.Q OR Refresh_Now THEN
			dly.PT := Refresh_Period;
			Refresh_Now := FALSE;
			state := START_READ;
		END_IF

	START_READ:(* === Start update when MB is free *)
		IF NOT (ModBus.MB_Lock OR ModBus.MB_Start) THEN

			ModBus.MB_Lock := TRUE;
			ModBus.MB_Query.SlaveAddress := Address;
			ModBus.MB_Query.FunctionCode := 16#03;
			(* Start query *)
			ModBus.MB_Query.Read_StartAddress := 16#0100;
			ModBus.MB_Query.Read_Quantity := 32;
			ModBus.MB_Start := TRUE;

			state := READ_1;
		END_IF

	READ_1:
		IF NOT ModBus.MB_Start THEN
			IF ModBus.MB_MASTER.MB_Error<>MB_NO_ERROR OR ModBus.MB_Resp.Error<>0 THEN
				state := ERROR_STATE;
			ELSE
				(* Read response data *)
				COPY_32SWAP16(ADR(ModBus.MB_Resp.Data[0]), ADR(Data.V_L1N));
				COPY_32SWAP16(ADR(ModBus.MB_Resp.Data[2]), ADR(Data.V_L2N));
				COPY_32SWAP16(ADR(ModBus.MB_Resp.Data[4]), ADR(Data.V_L3N));
				COPY_32SWAP16(ADR(ModBus.MB_Resp.Data[6]), ADR(Data.V_L1L2));
				COPY_32SWAP16(ADR(ModBus.MB_Resp.Data[8]), ADR(Data.V_L2L3));
				COPY_32SWAP16(ADR(ModBus.MB_Resp.Data[10]), ADR(Data.V_L3L1));
				COPY_32SWAP16(ADR(ModBus.MB_Resp.Data[12]), ADR(Data.I_L1));
				COPY_32SWAP16(ADR(ModBus.MB_Resp.Data[14]), ADR(Data.I_L2));
				COPY_32SWAP16(ADR(ModBus.MB_Resp.Data[16]), ADR(Data.I_L3));
				COPY_32SWAP16(ADR(ModBus.MB_Resp.Data[18]), ADR(Data.FREQ));
				COPY_32SWAP16(ADR(ModBus.MB_Resp.Data[20]), ADR(Data.P_3P));
				COPY_32SWAP16(ADR(ModBus.MB_Resp.Data[22]), ADR(Data.Q_3P));
				COPY_32SWAP16(ADR(ModBus.MB_Resp.Data[24]), ADR(Data.PF_3P));
				COPY_32SWAP16(ADR(ModBus.MB_Resp.Data[26]), ADR(Data.WH_3P));
				COPY_32SWAP16(ADR(ModBus.MB_Resp.Data[28]), ADR(Data.VARH_3P));
				COPY_32SWAP16(ADR(ModBus.MB_Resp.Data[28]), ADR(Data.Multiplier));

				(* Evaluate energy according to read multiplier factor *)
				WH_3P := (Data.WH_3P/100) * Data.Multiplier;		(* Divided by 100 because read value is in Wh, we need E-1 kWh *)
				VARH_3P := (Data.VARH_3P/100) * Data.Multiplier;

				ModBus.MB_Query.Read_StartAddress := 16#0122;
				ModBus.MB_Query.Read_Quantity := 4;
				ModBus.MB_Start := TRUE;

				state := READ_2;
			END_IF
		END_IF

	READ_2:
		IF NOT ModBus.MB_Start THEN
			IF ModBus.MB_MASTER.MB_Error<>MB_NO_ERROR OR ModBus.MB_Resp.Error<>0 THEN
				state := ERROR_STATE;
			ELSE
				(* Read response data *)
				COPY_32SWAP16(ADR(ModBus.MB_Resp.Data[0]), ADR(Data.V_3P));
				COPY_32SWAP16(ADR(ModBus.MB_Resp.Data[2]), ADR(Data.I_3P));

				ModBus.MB_Query.Read_StartAddress := 16#012E;
				ModBus.MB_Query.Read_Quantity := 2;
				ModBus.MB_Start := TRUE;

				state := READ_3;
			END_IF
		END_IF

	READ_3:
		IF NOT ModBus.MB_Start THEN
			IF ModBus.MB_MASTER.MB_Error<>MB_NO_ERROR OR ModBus.MB_Resp.Error<>0 THEN
				state := ERROR_STATE;
			ELSE
				(* Read response data *)
				COPY_32SWAP16(ADR(ModBus.MB_Resp.Data[0]), ADR(Data.COS_3P));

				ModBus.MB_Query.Read_StartAddress := 16#0142;
				ModBus.MB_Query.Read_Quantity := 20;
				ModBus.MB_Start := TRUE;

				state := READ_4;
			END_IF
		END_IF

	READ_4:
		IF NOT ModBus.MB_Start THEN
			IF ModBus.MB_MASTER.MB_Error<>MB_NO_ERROR OR ModBus.MB_Resp.Error<>0 THEN
				state := ERROR_STATE;
			ELSE
				COPY_32SWAP16(ADR(ModBus.MB_Resp.Data[0]), ADR(Data.VA_3P));
				COPY_32SWAP16(ADR(ModBus.MB_Resp.Data[2]), ADR(Data.P_L1));
				COPY_32SWAP16(ADR(ModBus.MB_Resp.Data[4]), ADR(Data.P_L2));
				COPY_32SWAP16(ADR(ModBus.MB_Resp.Data[6]), ADR(Data.P_L3));
				COPY_32SWAP16(ADR(ModBus.MB_Resp.Data[8]), ADR(Data.Q_L1));
				COPY_32SWAP16(ADR(ModBus.MB_Resp.Data[10]), ADR(Data.Q_L2));
				COPY_32SWAP16(ADR(ModBus.MB_Resp.Data[12]), ADR(Data.Q_L3));
				COPY_32SWAP16(ADR(ModBus.MB_Resp.Data[14]), ADR(Data.VA_L1));
				COPY_32SWAP16(ADR(ModBus.MB_Resp.Data[16]), ADR(Data.VA_L2));
				COPY_32SWAP16(ADR(ModBus.MB_Resp.Data[18]), ADR(Data.VA_L3));

				ModBus.MB_Query.Read_StartAddress := 16#0156;
				ModBus.MB_Query.Read_Quantity := 22;
				ModBus.MB_Start := TRUE;

				state := READ_5;
			END_IF
		END_IF

	READ_5:
		IF NOT ModBus.MB_Start THEN
			IF ModBus.MB_MASTER.MB_Error<>MB_NO_ERROR OR ModBus.MB_Resp.Error<>0 THEN
				state := ERROR_STATE;
			ELSE
				COPY_32SWAP16(ADR(ModBus.MB_Resp.Data[0]), ADR(Data.PF_L1));
				COPY_32SWAP16(ADR(ModBus.MB_Resp.Data[2]), ADR(Data.PF_L2));
				COPY_32SWAP16(ADR(ModBus.MB_Resp.Data[4]), ADR(Data.PF_L3));
				COPY_32SWAP16(ADR(ModBus.MB_Resp.Data[6]), ADR(Data.COS_L1));
				COPY_32SWAP16(ADR(ModBus.MB_Resp.Data[8]), ADR(Data.COS_L2));
				COPY_32SWAP16(ADR(ModBus.MB_Resp.Data[10]), ADR(Data.COS_L3));
				COPY_32SWAP16(ADR(ModBus.MB_Resp.Data[12]), ADR(Data.P_3P_Max));
				COPY_32SWAP16(ADR(ModBus.MB_Resp.Data[14]), ADR(Data.P_3P_Avg));
				COPY_32SWAP16(ADR(ModBus.MB_Resp.Data[16]), ADR(Data.I_L1_Max));
				COPY_32SWAP16(ADR(ModBus.MB_Resp.Data[18]), ADR(Data.I_L2_Max));
				COPY_32SWAP16(ADR(ModBus.MB_Resp.Data[20]), ADR(Data.I_L3_Max));

				ModBus.MB_Query.Read_StartAddress := 16#01A6;
				ModBus.MB_Query.Read_Quantity := 2;
				ModBus.MB_Start := TRUE;

				state := END_READ;
			END_IF
		END_IF

	END_READ:
		IF NOT ModBus.MB_Start THEN
			IF ModBus.MB_MASTER.MB_Error<>MB_NO_ERROR OR ModBus.MB_Resp.Error<>0 THEN
				state := ERROR_STATE;
			ELSE
				COPY_32SWAP16(ADR(ModBus.MB_Resp.Data[0]), ADR(Data.VA_3P));

				(* Signal event *)
				IF Status_Log<>0 THEN
					LogEv(EL_Log,EO_ANZ,ID,1,'');
				END_IF

				(* Update status *)
				Status_Log:=0;

				ModBus.MB_Lock := FALSE;
				retry := 0;
				state := WAIT_STATE;
			END_IF
		END_IF

	ERROR_STATE: (* === Check MODBUS error *)
			(* Release MODBUS *)
			MODBUS.MB_Lock:=FALSE;

			(* Retries *)
			retry:=retry+1;

			IF retry>3 THEN
				retry:=0;
				(* Signal event *)
				IF Status_Log<>2 THEN
					LogEv(EL_Alarm,EO_ANZ,ID,2,SEL(ModBus.MB_MASTER.MB_Error<>0,'0','1'));
				END_IF
				(* Update status *)
				Status_Log:=2;
			END_IF

			state := WAIT_STATE;

END_CASE

IF Status_Log=2 THEN Status_Vis := COLOR_RED;
ELSE Status_Vis := COLOR_GREEN;
END_IF
END_FUNCTION_BLOCK
ACTION AddLogData:
Logger.s1:=INSERT('&ANZ=',BYTE_TO_STRING(ID),4);
IF ID<10 THEN Logger.s1:=INSERT(Logger.s1,'0',4); END_IF

Logger.s1:=CONCAT(Logger.s1,DWORD_TO_STRING(Data.V_L1N/1000));		Logger.s1:=CONCAT(Logger.s1,';');
Logger.s1:=CONCAT(Logger.s1,DWORD_TO_STRING(Data.V_L2N/1000));		Logger.s1:=CONCAT(Logger.s1,';');
Logger.s1:=CONCAT(Logger.s1,DWORD_TO_STRING(Data.V_L3N/1000));		Logger.s1:=CONCAT(Logger.s1,';');
Logger.s1:=CONCAT(Logger.s1,DWORD_TO_STRING(Data.V_L1L2/1000));		Logger.s1:=CONCAT(Logger.s1,';');
Logger.s1:=CONCAT(Logger.s1,DWORD_TO_STRING(Data.V_L2L3/1000));		Logger.s1:=CONCAT(Logger.s1,';');
Logger.s1:=CONCAT(Logger.s1,DWORD_TO_STRING(Data.V_L3L1/1000));		Logger.s1:=CONCAT(Logger.s1,';');

Logger.s1:=CONCAT(Logger.s1,DWORD_TO_STRING(Data.FREQ));		Logger.s1:=CONCAT(Logger.s1,';');

Logger.s1:=CONCAT(Logger.s1,DWORD_TO_STRING(Data.I_L1));		Logger.s1:=CONCAT(Logger.s1,';');
Logger.s1:=CONCAT(Logger.s1,DWORD_TO_STRING(Data.I_L2));		Logger.s1:=CONCAT(Logger.s1,';');
Logger.s1:=CONCAT(Logger.s1,DWORD_TO_STRING(Data.I_L3));		Logger.s1:=CONCAT(Logger.s1,';');
Logger.s1:=CONCAT(Logger.s1,DWORD_TO_STRING(Data.I_L1_Max)); 	Logger.s1:=CONCAT(Logger.s1,';');
Logger.s1:=CONCAT(Logger.s1,DWORD_TO_STRING(Data.I_L2_Max)); 	Logger.s1:=CONCAT(Logger.s1,';');
Logger.s1:=CONCAT(Logger.s1,DWORD_TO_STRING(Data.I_L3_Max)); 	Logger.s1:=CONCAT(Logger.s1,';');

Logger.s1:=CONCAT(Logger.s1,DINT_TO_STRING(Data.PF_L1));		Logger.s1:=CONCAT(Logger.s1,';');
Logger.s1:=CONCAT(Logger.s1,DINT_TO_STRING(Data.PF_L2));		Logger.s1:=CONCAT(Logger.s1,';');
Logger.s1:=CONCAT(Logger.s1,DINT_TO_STRING(Data.PF_L3));		Logger.s1:=CONCAT(Logger.s1,';');

Logger.s1:=CONCAT(Logger.s1,DWORD_TO_STRING(Data.P_3P));		Logger.s1:=CONCAT(Logger.s1,';');
Logger.s1:=CONCAT(Logger.s1,DWORD_TO_STRING(Data.P_3P_Avg)); 	Logger.s1:=CONCAT(Logger.s1,';');
Logger.s1:=CONCAT(Logger.s1,DWORD_TO_STRING(Data.P_3P_Max)); 	Logger.s1:=CONCAT(Logger.s1,';');

Logger.s1:=CONCAT(Logger.s1,DWORD_TO_STRING(Data.Q_3P));		Logger.s1:=CONCAT(Logger.s1,';');
Logger.s1:=CONCAT(Logger.s1,DWORD_TO_STRING(Data.Q_3P_Max));	Logger.s1:=CONCAT(Logger.s1,';');

Logger.s1:=CONCAT(Logger.s1,DWORD_TO_STRING(WH_3P));		Logger.s1:=CONCAT(Logger.s1,';');
Logger.s1:=CONCAT(Logger.s1,DWORD_TO_STRING(VARH_3P));		Logger.s1:=CONCAT(Logger.s1,';');

Logger.s1:=CONCAT(Logger.s1,WORD_TO_STRING(Status_Log));
ADDSTRING(ADR(Logger.TData), ADR(Logger.s1), Logger.TLen);
END_ACTION

(* POU Plant_Objects/obj_MODBUS_TCP, ST *)
FUNCTION_BLOCK obj_MODBUS_TCP
(* === MODBUS-TCP PROTOCOL INTERFACE ===
   v1.0[10/06/15] - Create
*)
VAR CONSTANT
	VARS_Max	: BYTE := 32;
END_VAR
VAR_INPUT
	(* Settings *)
	ID			: BYTE;
	IP			: STRING;
	PORT		: WORD:=502;
	(* Interface *)
	MB_MASTER	: ETHERNET_MODBUSMASTER_TCP;
	MB_READBUF	: ARRAY [0..128] OF WORD;
	MB_WRITEBUF : ARRAY [0..128] OF WORD;
	MB_Start	: BOOL;
	MB_Lock		: BOOL;
	(* Variables management *)
	VARS_En		: BOOL;
	VARS		: ARRAY [0..VARS_Max] OF typ_MODBUS_VAR;
	VARS_Check	: BOOL;
	VARS_Alarm	: BOOL;
	(* Variables allocation *)
	VAR_Pointer : POINTER TO ARRAY[0..99] OF WORD;
	VAR_Cfg		: POINTER TO typ_MODBUS_VAR;
END_VAR
VAR_OUTPUT
	(* Status *)
	Status_Log	: BYTE;
	Status_Vis	: DWORD;
END_VAR
VAR
	sta         : BYTE :=0;
	i			: BYTE;
	j			: BYTE;
	Alarm		: FLT_EVENT;

	VarTmr		: TON := (PT:=T#1s);
	VarSta		: BYTE; (* Status *)
	VarCnt		: BYTE; (* Scan counter *)
	VarRetry	: BYTE;
	VarAlarm	: BYTE; (* Last variable with errors *)
END_VAR
MB_MASTER( strIP_ADDRESS:=IP, wPORT:=PORT, tTIME_OUT:=T#750MS, (*xCONNECT:=TRUE,*)
		   ptREAD_DATA:=ADR(MB_READBUF), ptSEND_DATA:=ADR(MB_WRITEBUF), xSEND:=MB_Start );

IF sta=0 THEN
	MB_MASTER.xCONNECT:=TRUE;
	sta:=1;
END_IF

(* Process variable management *)
IF VARS_En THEN VARS_Process(); END_IF

(* Check status *)
Alarm(IN:=(MB_MASTER.wERROR<>0));
IF Alarm.EVH THEN
	LogEv(SEL(MB_MASTER.wERROR>0,EL_Wrn,EL_Alarm),EO_MODBUS_TCP,ID,1,WORD_TO_STRING(MB_MASTER.wERROR));
END_IF
IF Alarm.EVL THEN
	LogEv(EL_Log,EO_MODBUS_TCP,ID,2,'');
END_IF

(* Log/visu status *)
   IF Alarm.IN   THEN Status_Log:=2; Status_Vis:=COLOR_RED;
ELSIF Vars_Alarm THEN Status_Log:=1; Status_Vis:=COLOR_YELLOW;
  				 ELSE Status_Log:=0; Status_Vis:=COLOR_GREEN;
END_IF
END_FUNCTION_BLOCK
ACTION VAR_Search:
(* Search VAR with specific pointer if not found return first free VAR
	[Last VAR is not active... used as safe area...] 
*)
j:=VARS_Max;
FOR i := 0 TO VARS_Max-1 DO
	IF VARS[i].Variable=0 AND j>i THEN j:=i; END_IF
	IF VARS[i].Variable=VAR_Pointer THEN
		VAR_Cfg:=ADR(VARS[i]);
		RETURN;
	END_IF
END_FOR
VAR_Cfg:=ADR(VARS[j]);
END_ACTION
ACTION VARS_Process:
(* Update var timers *)
VarTmr(IN:=(NOT VarTmr.Q));
IF VarTmr.Q THEN
	FOR i := 0 TO VARS_Max DO
		IF VARS[i].Refresh_Cnt>0 THEN VARS[i].Refresh_Cnt:=VARS[i].Refresh_Cnt-1; END_IF
	END_FOR
	VARS_Check:=TRUE;
END_IF


(* Process status *)
CASE VarSta OF
	0: (* === Init *)
		VarCnt:=0;
		VarSta:=1;

	1: (* === Wait check signal *)
		IF VARS_Check THEN
			VARS_Check:=FALSE;
			VarCnt:=0;
			VarSta:=2;
		END_IF

	2: (* === Check loop *)
		IF NOT (MB_Lock OR MB_Start) THEN
			WHILE VarCnt<=(VARS_Max-1) AND VarSta=2 DO
				(* Check only active vars *)
				IF VARS[VarCnt].Variable<>0 THEN
					(* Check var auto-refresh on timer checks *)
					IF VARS[VarCnt].Refresh_Time>0 AND VARS[VarCnt].Refresh_Cnt=0 THEN
						VARS[VarCnt].Refresh_Cnt:=VARS[VarCnt].Refresh_Time;
						VarSta:=3;
					END_IF
					(* Check refresh for change or request *)
					CASE VARS[VarCnt].FunCode OF
						5,6,15,16: (* Write functions *)
							IF VARS[VarCnt].Variable_Size=1 THEN
								IF VARS[VarCnt].Variable^<>VARS[VarCnt].Variable_Mirror THEN
									VARS[VarCnt].Variable_Mirror:=VARS[VarCnt].Variable^;
									VarSta:=3;
								END_IF
							ELSE
								IF VARS[VarCnt].Variable_Mirror<>0 THEN
									VARS[VarCnt].Variable_Mirror:=0;
									VarSta:=3;
								END_IF
							END_IF
						1,2,3,4: (* Write functions *)
							IF VARS[VarCnt].Variable_Mirror<>0 THEN
								VARS[VarCnt].Variable_Mirror:=0;
								VarSta:=3;
							END_IF
					END_CASE
				END_IF
				(* Process query *)
				IF VarSta=3 THEN
					MB_Lock:=TRUE;
					MB_MASTER.bUNIT_ID:=VARS[VarCnt].SlaveAddress;
					MB_MASTER.bFUNCTION_CODE:=VARS[VarCnt].FunCode;
					CASE VARS[VarCnt].FunCode OF
						16#5,16#6,16#F,16#10:
							MB_MASTER.wREAD_ADDRESS:=0;
							MB_MASTER.wREAD_QUANTITY:=0;
							MB_MASTER.wWRITE_ADDRESS:=VARS[VarCnt].FunAddress;
							MB_MASTER.wWRITE_QUANTITY:=VARS[VarCnt].Variable_Size;
							IF VARS[VarCnt].Variable_Size=200 THEN
								COPY_32SWAP16(VARS[VarCnt].Variable, ADR(MB_WRITEBUF));
							ELSIF VARS[VarCnt].Variable_Size>1 THEN
								MEMCPY(VARS[VarCnt].Variable, ADR(MB_WRITEBUF), 2*VARS[VarCnt].Variable_Size);
							ELSE
								MB_WRITEBUF[0]:=VARS[VarCnt].Variable^;
							END_IF
						16#1,16#2,16#3,16#4:
							MB_MASTER.wREAD_ADDRESS:=VARS[VarCnt].FunAddress;
							IF VARS[VarCnt].Variable_Size=200 THEN MB_MASTER.wREAD_QUANTITY:=2; ELSE
							  MB_MASTER.wREAD_QUANTITY:=VARS[VarCnt].Variable_Size;
							END_IF
							MB_MASTER.wWRITE_ADDRESS:=0;
							MB_MASTER.wWRITE_QUANTITY:=0;
					END_CASE
					VarRetry:=0;
					MB_Start:=TRUE;
				ELSE
					VarCnt:=VarCnt+1;
				END_IF
			END_WHILE
			(* Check loop completed -> no actions *)
			IF VarSta=2 THEN VarSta:=1; END_IF
		END_IF

	3: (* === Wait & process MB response *)
		IF NOT MB_Start THEN
			IF MB_MASTER.wERROR=0 THEN
				CASE VARS[VarCnt].FunCode OF
					1,2,3,4:
						IF VARS[VarCnt].Variable_Size=200 THEN
							COPY_32SWAP16(ADR(MB_READBUF), VARS[VarCnt].Variable);
						ELSIF VARS[VarCnt].Variable_Size>1 THEN
							MEMCPY(ADR(MB_READBUF), VARS[VarCnt].Variable, 2*VARS[VarCnt].Variable_Size);
						ELSE
							VARS[VarCnt].Variable^:=MB_READBUF[0];
						END_IF
				END_CASE
				MB_Lock:=FALSE;
				(* Signal error recovery *)
				IF VARS_Alarm=TRUE AND VarCnt=VarAlarm THEN
					LogEv(EL_Wrn,EO_MODBUS_TCP,ID,5,'');
					VARS_Alarm:=FALSE;
				END_IF
				(* Next var *)
				VarCnt:=VarCnt+1;
				VarSta:=2;
			ELSE
				IF VarRetry<10 THEN
					VarRetry:=VarRetry+1;
					MB_Start:=TRUE;
				ELSE
					MB_Lock:=FALSE;
					(* Signal error *)
					IF VARS_Alarm=FALSE THEN
						LogEv(EL_Wrn,EO_MODBUS_TCP,ID,3,WORD_TO_STRING(MB_MASTER.wERROR));
						VARS_Alarm:=TRUE;
						VarAlarm:=VarCnt-1;
					END_IF
					(* Next var *)
					VarCnt:=VarCnt+1;
					VarSta:=2;
				END_IF
			END_IF
		END_IF

ELSE
	VarSta:=0;
END_CASE
END_ACTION

(* POU Plant_Objects/obj_ZTHL, ST *)
FUNCTION_BLOCK obj_ZTHL
(* === ZIGBEE AMBIENT SENSORS MT-200 ===
   v1.0[07/05/05] - Create
*)
VAR CONSTANT
	(* States *)
	WAIT_STATE			:	BYTE := 0;
	STATUS_REQUEST		:	BYTE := 1;
	LQI_REQUEST			:	BYTE := 2;
	MEAS_REQUEST		:	BYTE := 3;
	END_READ			:	BYTE := 4;
	ERROR_STATE			:	BYTE := 100;

	LQI_Threshold		:	WORD := 100;		(* Zigbee link quality minimum value *)
	LowBattVoltage		:	WORD := 270;		(* Battery is considered low when reaches 1.35V each *)
END_VAR
VAR_INPUT
	(* Settings *)
	ID				: BYTE;
	Address			: BYTE;

	Refresh_Period	: TIME:=t#5m;
	(* Controls *)
	Refresh_Auto	: BOOL:=TRUE; (* Enable automatic refresh *)
	Refresh_Now		: BOOL; 	  (* Force an immediate refresh *)

	(* Limits *)
	Tmin			: INT := 0;
	Tmax			: INT := 400;
END_VAR
VAR_IN_OUT
	(* Interface *)
	MODBUS			: obj_MODBUS_TCP;
END_VAR
VAR_OUTPUT
	OUT_TEMP		: INT;	(* Temperatura misurata [°C/10] *)
	OUT_HYGRO		: INT;	(* Umidità misurata [%] *)
	OUT_LUX			: INT;	(* Luce misurata [lux] *)
	OUT_VBATT		: INT;	(* Tensione misurata dalla batteria [V/100] *)

	OUT_LQI			: BYTE;

	ERR				: BOOL;

	fTemp			: BOOL;

	(* Status *)
	Status_Log		: BYTE;
	Status_Vis 		: DWORD;
END_VAR
VAR
	dly 	 		: TON := (PT:=t#5s);

	sta				: BYTE;
	retry	 		: BYTE;

	OldNodeStatus	: WORD;
	fLQI			: BOOL;
	fBatt			: BOOL;
	Quality			: FLT_EVENT;
	Battery			: FLT_EVENT;
	Temperature		: FLT_EVENT;
	Alarm			: FLT_EVENT;

	StatusOK		: BYTE;			(* 0: Status OK, >=1: Alarm and/or warning		Incremented by 1 when Alarm or Wrn occurs,
																					decremented by 1 when restored	*)
END_VAR
CASE sta OF
	WAIT_STATE: (* === Wait update signals *)
		dly(IN:=NOT (dly.Q OR Refresh_Now OR (NOT Refresh_Auto)));
		IF dly.Q OR Refresh_Now THEN
			dly.PT:=Refresh_Period;
			Refresh_Now:=FALSE;
			(*sta:=STATUS_REQUEST;*)
			sta:=LQI_REQUEST;
		END_IF

	STATUS_REQUEST:	(* Node status *)
		IF NOT (MODBUS.MB_Lock OR MODBUS.MB_Start) THEN
			MODBUS.MB_Lock:=TRUE;
			MODBUS.ID:=ID;
			MODBUS.MB_MASTER.bUNIT_ID := Address;
			MODBUS.MB_MASTER.bFUNCTION_CODE:=16#03;
			MODBUS.MB_MASTER.wREAD_ADDRESS:=16#0D;
			MODBUS.MB_MASTER.wREAD_QUANTITY:=16#1;
			MODBUS.MB_Start:=TRUE;
			sta:=LQI_REQUEST;
		END_IF

	LQI_REQUEST:	(* Link quality *)
		IF NOT MODBUS.MB_Start THEN
			IF MODBUS.MB_MASTER.wERROR<>MB_NO_ERROR THEN
				sta:=ERROR_STATE;
			ELSE
				(*NodeStatus	:=	MODBUS.MB_READBUF[0];*)

				MODBUS.ID:=ID;
				MODBUS.MB_MASTER.bUNIT_ID := Address;
				MODBUS.MB_MASTER.bFUNCTION_CODE:=16#03;
				MODBUS.MB_MASTER.wREAD_ADDRESS:=16#01;
				MODBUS.MB_MASTER.wREAD_QUANTITY:=16#1;
				MODBUS.MB_Start:=TRUE;

				sta:=MEAS_REQUEST;
			END_IF
		END_IF

	MEAS_REQUEST:	(* Measurements *)
		IF NOT MODBUS.MB_Start THEN
			IF MODBUS.MB_MASTER.wERROR<>MB_NO_ERROR THEN
				sta:=ERROR_STATE;
			ELSE

				OUT_LQI	:=	WORD_TO_BYTE(MODBUS.MB_READBUF[0]);

				MODBUS.ID:=ID;
				MODBUS.MB_MASTER.bUNIT_ID := Address;
				MODBUS.MB_MASTER.bFUNCTION_CODE:=16#03;
				MODBUS.MB_MASTER.wREAD_ADDRESS:=16#14;
				MODBUS.MB_MASTER.wREAD_QUANTITY:=16#5;
				MODBUS.MB_Start:=TRUE;

				sta:=END_READ;
			END_IF
		END_IF

	END_READ:	IF NOT MODBUS.MB_Start THEN
			IF MODBUS.MB_MASTER.wERROR<>MB_NO_ERROR THEN
				sta:=ERROR_STATE;
			ELSE
				OUT_TEMP	:=	WORD_TO_INT(MODBUS.MB_READBUF[0]);
				OUT_HYGRO	:=	WORD_TO_INT(MODBUS.MB_READBUF[1]);
				OUT_LUX		:=	WORD_TO_INT(MODBUS.MB_READBUF[2]);
				OUT_VBATT	:=	WORD_TO_INT(MODBUS.MB_READBUF[3]);
				sta:=WAIT_STATE;
				MODBUS.MB_Lock:=FALSE;
			END_IF
		END_IF

	ERROR_STATE:
			MODBUS.MB_Lock:=FALSE;
			(* Retries *)
			retry:=retry+1;
			IF retry>3 THEN
				retry:=0;
				IF Status_Log<>2 THEN
					LogEv(EL_Alarm,EO_ZTHL,ID,4,'');
				END_IF
				Status_Log:=2;
				Status_Vis:=COLOR_RED;
			END_IF
			sta:=WAIT_STATE;

ELSE
			sta:=WAIT_STATE;
END_CASE

(* Check Status *)
(*
IF NodeStatus <> OldNodeStatus THEN
	IF NodeStatus = 3 THEN
		LogEv(EL_Alarm,EO_ZTHL,ID,3,'');
		Status_Log:=2;
	ELSE
		Status_Log:=0;
	END_IF

	OldNodeStatus := NodeStatus;
END_IF*)

(* Check Link quality *)
IF OUT_LQI > LQI_Threshold THEN
	fLQI := TRUE;
	ERR := TRUE;
ELSE
	fLQI := FALSE;
	ERR := FALSE;
END_IF

Quality(IN:=fLQI);

IF Quality.EVL THEN
	LogEv(SEL(OUT_LQI<>0,EL_Alarm,EL_Wrn),EO_ZTHL,ID,SEL(OUT_LQI<>0,7,2),WORD_TO_STRING(OUT_LQI));
	Status_Log := SEL(OUT_LQI<>0,2,1);
	StatusOK := StatusOK + 1;
END_IF

IF Quality.EVH THEN StatusOK := SEL(StatusOK=0, StatusOK-1, 0); END_IF

(* If probe (node) is present proceed checking other warnings, otherwise don't transmit anything *)
IF OUT_LQI <> 0 THEN

	(* Check battery voltage *)
	IF OUT_VBATT < LowBattVoltage THEN fBatt := TRUE;
	ELSE fBatt := FALSE;
	END_IF
	
	Battery(IN:=fBatt);
	
	IF Battery.EVH THEN
		LogEv(EL_Wrn,EO_ZTHL,ID,6,'');
		StatusOK := StatusOK + 1;
	END_IF

	IF Battery.EVL THEN StatusOK := SEL(StatusOK=0, StatusOK-1, 0); END_IF

	(* Check Node temperature *)
	IF OUT_TEMP < Tmin OR OUT_TEMP > Tmax THEN
		fTemp := TRUE;
		ERR := TRUE;
	ELSE
		fTemp := FALSE;
		ERR := FALSE;
	END_IF

	Temperature(IN:=fTemp);

	IF Temperature.EVH THEN
		LogEv(EL_Wrn,EO_ZTHL,ID,5,INT_TO_STRING(OUT_TEMP));
		Status_Log := 1;
		StatusOK := StatusOK + 1;
	END_IF

	IF Temperature.EVL THEN StatusOK := SEL(StatusOK=0, StatusOK-1, 0); END_IF

END_IF

Alarm(IN:=(StatusOK=0));

IF Alarm.EVH THEN
	Status_Log := 0;
	LogEv(EL_Log,EO_ZTHL,ID,1,'');
END_IF

IF Status_Log = 2 THEN Status_Vis := COLOR_RED;
ELSIF Status_Log = 1 THEN Status_Vis := COLOR_YELLOW;
ELSE Status_Vis := COLOR_GREEN;
END_IF
END_FUNCTION_BLOCK
ACTION AddLogData:
Logger.s1:=INSERT('&ZTHL=',BYTE_TO_STRING(ID),5);
IF ID<10 THEN Logger.s1:=INSERT(Logger.s1,'0',4); END_IF

Logger.s1:=CONCAT(Logger.s1,BYTE_TO_STRING(OUT_LQI));			Logger.s1:=CONCAT(Logger.s1,';');
Logger.s1:=CONCAT(Logger.s1,INT_TO_STRING(OUT_TEMP ));			Logger.s1:=CONCAT(Logger.s1,';');
Logger.s1:=CONCAT(Logger.s1,INT_TO_STRING(OUT_HYGRO ));			Logger.s1:=CONCAT(Logger.s1,';');
Logger.s1:=CONCAT(Logger.s1,INT_TO_STRING(OUT_LUX));			Logger.s1:=CONCAT(Logger.s1,';');
Logger.s1:=CONCAT(Logger.s1,INT_TO_STRING(OUT_VBATT));			Logger.s1:=CONCAT(Logger.s1,';');

Logger.s1:=CONCAT(Logger.s1,BYTE_TO_STRING(Status_Log));
ADDSTRING(ADR(Logger.TData), ADR(Logger.s1), Logger.TLen);
END_ACTION

(* POU PLC_WDT, ST *)
FUNCTION PLC_WDT: DWORD VAR_INPUT dwEvent: DWORD; dwFilter: DWORD; dwOwner: DWORD; END_VAR
LogEv(EL_AlarmStop,EO_SYS,1,10,'Watchdog');
END_FUNCTION

(* POU Utils Functions/RAWTOHEXSTR, ST *)
FUNCTION RAWTOHEXSTR : STRING(128)
VAR_INPUT
	pData: POINTER TO BYTE;
	DataLen: BYTE;
END_VAR
VAR
	pt: POINTER TO BYTE;
	xl: BYTE;
END_VAR
pt:=ADR(RAWTOHEXSTR);

xl:=2;

WHILE DataLen>0 AND xl<128 DO

	pt^ := (pData^ / 16#10) + 48 + (((pData^ / 16#10)/10)*7);
	pt:=pt+1;
	pt^ := (pData^ AND 16#0F)  + 48 + (((pData^ AND 16#0F)/10)*7);
	pt:=pt+1;

	xl:=xl+2;

	DataLen:=DataLen-1;
	pData:=pData+1;

END_WHILE

pt^:=0;
END_FUNCTION

(* POU Utils Functions/RESET_ARRAY, ST *)
FUNCTION RESET_ARRAY : BOOL
VAR_INPUT
	pData	:	POINTER TO WORD;
	Size	:	BYTE;
END_VAR
VAR
	i	:	BYTE := 0;
END_VAR
WHILE i<Size DO

	pData^ := 0;
	pData := pData + 1;
	i := i + 1;

END_WHILE
END_FUNCTION

(* POU Utils/RTC_Update, ST *)
FUNCTION RTC_Update : BOOL
VAR
	T: DT;
	TS: STRING;
	TS2: STRING;
	Hour: BYTE;
	Minute: BYTE;
END_VAR
(* Get RTC time *)
T:=SysRtcGetTime(TRUE);
Sys.Time_CT_DT:=T;
(* Calculate variables *)
TS:=DT_TO_STRING(T);
Sys.Time_LogString:=DELETE(STR:=TS, LEN:=3, POS:=1);
TS2:=MID(STR:=TS, LEN:=4, POS:= 4); Sys.Time_Year 	:=STRING_TO_WORD(TS2);
TS2:=MID(STR:=TS, LEN:=2, POS:= 9); Sys.Time_Month	:=STRING_TO_BYTE(TS2);
TS2:=MID(STR:=TS, LEN:=2, POS:=12); Sys.Time_Day  	:=STRING_TO_BYTE(TS2);
Sys.Time_CT_Day:=(32*(Sys.Time_Month-1)+Sys.Time_Day-1);
TS2:=MID(STR:=TS, LEN:=2, POS:=15); Hour			:=STRING_TO_BYTE(TS2);
TS2:=MID(STR:=TS, LEN:=2, POS:=18); Minute		 	:=STRING_TO_BYTE(TS2);
Sys.Time_CT_Quarter:=Hour*4+(Minute/15);
END_FUNCTION

(* POU Utils Functions/SHIFT_ARRAY, ST *)
FUNCTION SHIFT_ARRAY : BOOL
VAR_INPUT
	pData	:	POINTER TO WORD;
	Size	:	BYTE;
END_VAR
VAR
	pNew	:	POINTER TO WORD;
	i		:	BYTE;
END_VAR
(* Shift right *)
FOR i:=1 TO (Size-1) BY 1 DO

	pNew := pData + 1;
	pData^ := pNew^;
	pData := pData + 1;

	i := i + 1;
END_FOR
END_FUNCTION

(* POU Utils Functions/TONOF, ST *)
FUNCTION_BLOCK TONOF
VAR_INPUT
	IN		: BOOL;
	PT_ON	: TIME; (* time to pass, before OUT is set *)
	PT_OF	: TIME; (* time to pass, before OUT is reset *)
END_VAR
VAR_OUTPUT
	OUT		: BOOL;
END_VAR
VAR
	timer	: TON;
END_VAR
IF IN<>OUT THEN
	timer(IN:=TRUE,PT:=SEL(IN,PT_OF,PT_ON));
	IF timer.Q THEN OUT:=IN; END_IF
ELSE
	timer(IN:=FALSE);
END_IF
END_FUNCTION_BLOCK

(* Visualisation PLC_VISU
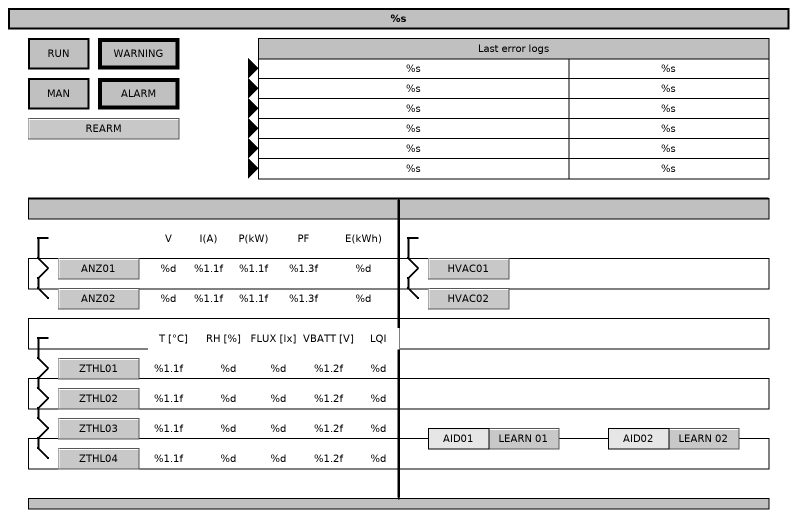
rectangle at (10,0)-(791,21): text "%s"; shows .Plant_NAME
rounded rectangle at (30,30)-(91,61): text "RUN"; alarm colour if NOT Mode_Manual; runs INTERN ASSIGN Mode_Manual:=(FALSE)
rounded rectangle at (30,70)-(91,101): text "MAN"; alarm colour if Mode_Manual; runs INTERN ASSIGN Mode_Manual:=(TRUE)
rectangle at (570,50)-(771,71): text "%s"; shows Sys.LastLogs_Msg[0]
polygon at (250,150)-(260,170): invisible if Sys.LastLogs_Idx<>0
rectangle at (570,70)-(771,91): text "%s"; shows Sys.LastLogs_Msg[1]
polygon at (250,50)-(260,70): invisible if Sys.LastLogs_Idx<>1
rectangle at (570,90)-(771,111): text "%s"; shows Sys.LastLogs_Msg[2]
polygon at (250,70)-(260,90): invisible if Sys.LastLogs_Idx<>2
rectangle at (570,110)-(771,131): text "%s"; shows Sys.LastLogs_Msg[3]
polygon at (250,90)-(260,110): invisible if Sys.LastLogs_Idx<>3
rectangle at (570,130)-(771,151): text "%s"; shows Sys.LastLogs_Msg[4]
polygon at (250,110)-(260,130): invisible if Sys.LastLogs_Idx<>4
rectangle at (570,150)-(771,171): text "%s"; shows Sys.LastLogs_Msg[5]
polygon at (250,130)-(260,150): invisible if Sys.LastLogs_Idx<>5
rectangle at (260,50)-(571,71): text "%s"; shows Sys.LastLogs_Dat[0]
rectangle at (260,70)-(571,91): text "%s"; shows Sys.LastLogs_Dat[1]
rectangle at (260,90)-(571,111): text "%s"; shows Sys.LastLogs_Dat[2]
rectangle at (260,110)-(571,131): text "%s"; shows Sys.LastLogs_Dat[3]
rectangle at (260,130)-(571,151): text "%s"; shows Sys.LastLogs_Dat[4]
rectangle at (260,150)-(571,171): text "%s"; shows Sys.LastLogs_Dat[5]
rectangle at (100,70)-(181,101): text "ALARM"; alarm colour if Sys.Alarm; runs INTERN ASSIGN Mode_Manual:=(FALSE)
rectangle at (100,30)-(181,61): text "WARNING"; alarm colour if Sys.Warning; runs INTERN ASSIGN Mode_Manual:=(TRUE)
button at (30,110)-(181,131): text "REARM"; runs INTERN ASSIGN Sys.Alarm:=(FALSE);INTERN ASSIGN Sys.Warning:=(FALSE)
button at (60,250)-(141,271): text "ANZ01"
rectangle at (260,30)-(771,51): text "Last error logs"
button at (60,280)-(141,301): text "ANZ02"
rectangle at (150,220)-(191,241): text "V"
rectangle at (230,220)-(281,241): text "P(kW)"
rectangle at (280,220)-(331,241): text "PF"
rectangle at (330,220)-(401,241): text "E(kWh)"
rectangle at (190,220)-(231,241): text "I(A)"
rectangle at (150,250)-(191,271): text "%d"; shows ANZ01.Data.V_3P/1000
rectangle at (190,250)-(231,271): text "%1.1f"; shows DWORD_TO_REAL(ANZ01.Data.I_3P)/1000
rectangle at (230,250)-(281,271): text "%1.1f"; shows DWORD_TO_REAL(ANZ01.Data.P_3P)/1000
rectangle at (280,250)-(331,271): text "%1.3f"; shows DINT_TO_REAL(ANZ01.Data.PF_3P)/1000
rectangle at (330,250)-(401,271): text "%d"; shows ANZ01.WH_3P/10
rectangle at (150,280)-(191,301): text "%d"; shows ANZ02.Data.V_3P/1000
rectangle at (190,280)-(231,301): text "%1.1f"; shows DWORD_TO_REAL(ANZ02.Data.I_3P)/1000
rectangle at (230,280)-(281,301): text "%1.1f"; shows DWORD_TO_REAL(ANZ02.Data.P_3P)/1000
rectangle at (280,280)-(331,301): text "%1.3f"; shows DINT_TO_REAL(ANZ02.Data.PF_3P)/1000
rectangle at (330,280)-(401,301): text "%d"; shows ANZ02.WH_3P/10
button at (430,250)-(511,271): text "HVAC01"
button at (430,280)-(511,301): text "HVAC02"
button at (490,420)-(561,441): text "LEARN 01"; runs INTERN ASSIGN AID01.Status:=(1)
button at (670,420)-(741,441): text "LEARN 02"; runs INTERN ASSIGN AID02.Status:=(1)
rectangle at (430,420)-(491,441): text "AID01"
rectangle at (610,420)-(671,441): text "AID02"
button at (60,350)-(141,371): text "ZTHL01"
button at (60,380)-(141,401): text "ZTHL02"
button at (60,410)-(141,431): text "ZTHL03"
button at (60,440)-(141,461): text "ZTHL04"
rectangle at (150,350)-(191,371): text "%1.1f"; shows INT_TO_REAL(ZTHL01.OUT_TEMP)/10
rectangle at (150,320)-(201,341): text "T [°C]"
rectangle at (200,320)-(251,341): text "RH [%]"
rectangle at (250,320)-(301,341): text "FLUX [lx]"
rectangle at (300,320)-(361,341): text "VBATT [V]"
rectangle at (360,320)-(401,341): text "LQI"
rectangle at (210,350)-(251,371): text "%d"; shows ZTHL01.OUT_HYGRO
rectangle at (260,350)-(301,371): text "%d"; shows ZTHL01.OUT_LUX
rectangle at (310,350)-(351,371): text "%1.2f"; shows INT_TO_REAL(ZTHL01.OUT_VBATT)/100
rectangle at (360,350)-(401,371): text "%d"; shows ZTHL01.OUT_LQI
rectangle at (150,380)-(191,401): text "%1.1f"; shows INT_TO_REAL(ZTHL02.OUT_TEMP)/10
rectangle at (210,380)-(251,401): text "%d"; shows ZTHL02.OUT_HYGRO
rectangle at (260,380)-(301,401): text "%d"; shows ZTHL02.OUT_LUX
rectangle at (310,380)-(351,401): text "%1.2f"; shows INT_TO_REAL(ZTHL02.OUT_VBATT)/100
rectangle at (360,380)-(401,401): text "%d"; shows ZTHL02.OUT_LQI
rectangle at (150,410)-(191,431): text "%1.1f"; shows INT_TO_REAL(ZTHL03.OUT_TEMP)/10
rectangle at (210,410)-(251,431): text "%d"; shows ZTHL03.OUT_HYGRO
rectangle at (260,410)-(301,431): text "%d"; shows ZTHL03.OUT_LUX
rectangle at (310,410)-(351,431): text "%1.2f"; shows INT_TO_REAL(ZTHL03.OUT_VBATT)/100
rectangle at (360,410)-(401,431): text "%d"; shows ZTHL03.OUT_LQI
rectangle at (150,440)-(191,461): text "%1.1f"; shows INT_TO_REAL(ZTHL04.OUT_TEMP)/10
rectangle at (210,440)-(251,461): text "%d"; shows ZTHL04.OUT_HYGRO
rectangle at (260,440)-(301,461): text "%d"; shows ZTHL04.OUT_LUX
rectangle at (310,440)-(351,461): text "%1.2f"; shows INT_TO_REAL(ZTHL04.OUT_VBATT)/100
rectangle at (360,440)-(401,461): text "%d"; shows ZTHL04.OUT_LQI
16 more shapes without text or variables
18 elements of other kinds (tables, trends, ...) not read
*)

